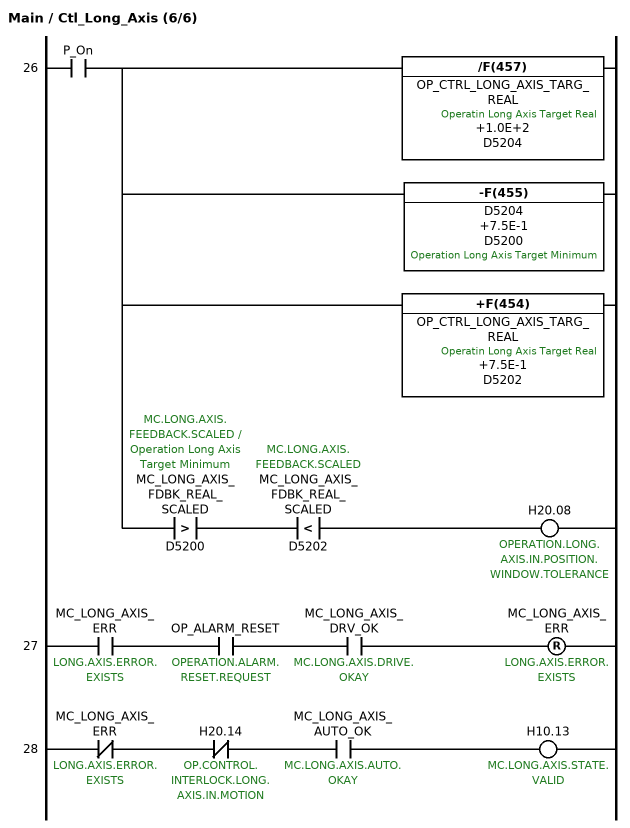
; [picture p48: Main / Ctl_Long_Axis, rungs 26-28]
; rung 26
LD P_On
/F(457) OP_CTRL_LONG_AXIS_TARG_REAL +1.0E+2 D5204  ; Operatin Long Axis Target Real
-F(455) D5204 +7.5E-1 D5200  ; Operation Long Axis Target Minimum
+F(454) OP_CTRL_LONG_AXIS_TARG_REAL +7.5E-1 D5202  ; Operatin Long Axis Target Real
AND>F(333) MC_LONG_AXIS_FDBK_REAL_SCALED D5200  ; MC.LONG.AXIS.FEEDBACK.SCALED, Operation Long Axis Target Minimum
AND<F(331) MC_LONG_AXIS_FDBK_REAL_SCALED D5202  ; MC.LONG.AXIS.FEEDBACK.SCALED
OUT H20.08  ; OPERATION.LONG.AXIS.IN.POSITION.WINDOW.TOLERANCE
; rung 27
LD MC_LONG_AXIS_ERR  ; LONG.AXIS.ERROR.EXISTS
AND OP_ALARM_RESET  ; OPERATION.ALARM.RESET.REQUEST
AND MC_LONG_AXIS_DRV_OK  ; MC.LONG.AXIS.DRIVE.OKAY
RSET MC_LONG_AXIS_ERR  ; LONG.AXIS.ERROR.EXISTS
; rung 28
LDNOT MC_LONG_AXIS_ERR  ; LONG.AXIS.ERROR.EXISTS
ANDNOT H20.14  ; OP.CONTROL.INTERLOCK.LONG.AXIS.IN.MOTION
AND MC_LONG_AXIS_AUTO_OK  ; MC.LONG.AXIS.AUTO.OKAY
OUT H10.13  ; MC.LONG.AXIS.STATE.VALID

### Section Ctl_Vertical_Axis

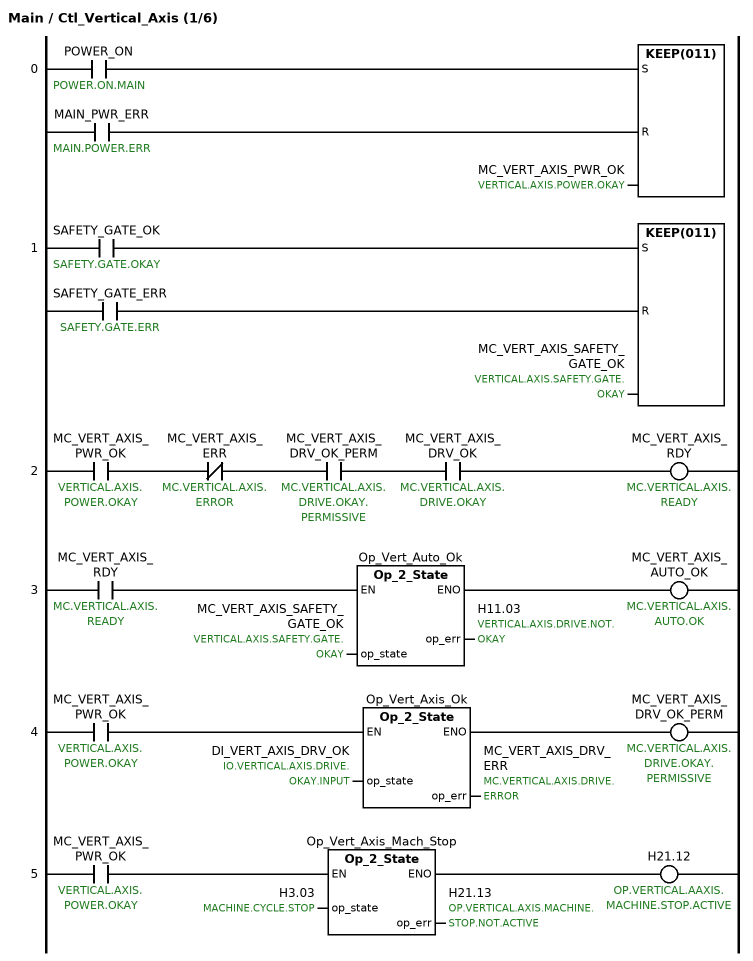
; rung 0
LD POWER_ON  ; POWER.ON.MAIN
LD MAIN_PWR_ERR  ; MAIN.POWER.ERR
KEEP(011) MC_VERT_AXIS_PWR_OK  ; VERTICAL.AXIS.POWER.OKAY
; rung 1
LD SAFETY_GATE_OK  ; SAFETY.GATE.OKAY
LD SAFETY_GATE_ERR  ; SAFETY.GATE.ERR
KEEP(011) MC_VERT_AXIS_SAFETY_GATE_OK  ; VERTICAL.AXIS.SAFETY.GATE.OKAY
; rung 2
LD MC_VERT_AXIS_PWR_OK  ; VERTICAL.AXIS.POWER.OKAY
ANDNOT MC_VERT_AXIS_ERR  ; MC.VERTICAL.AXIS.ERROR
AND MC_VERT_AXIS_DRV_OK_PERM  ; MC.VERTICAL.AXIS.DRIVE.OKAY.PERMISSIVE
AND MC_VERT_AXIS_DRV_OK  ; MC.VERTICAL.AXIS.DRIVE.OKAY
OUT MC_VERT_AXIS_RDY  ; MC.VERTICAL.AXIS.READY
; rung 3
LD MC_VERT_AXIS_RDY  ; MC.VERTICAL.AXIS.READY
CALL Op_Vert_Auto_Ok : Op_2_State (op_state := MC_VERT_AXIS_SAFETY_GATE_OK, op_err => H11.03)  ; VERTICAL.AXIS.SAFETY.GATE.OKAY, VERTICAL.AXIS.DRIVE.NOT.OKAY
OUT MC_VERT_AXIS_AUTO_OK  ; MC.VERTICAL.AXIS.AUTO.OK
; rung 4
LD MC_VERT_AXIS_PWR_OK  ; VERTICAL.AXIS.POWER.OKAY
CALL Op_Vert_Axis_Ok : Op_2_State (op_state := DI_VERT_AXIS_DRV_OK, op_err => MC_VERT_AXIS_DRV_ERR)  ; IO.VERTICAL.AXIS.DRIVE.OKAY.INPUT, MC.VERTICAL.AXIS.DRIVE.ERROR
OUT MC_VERT_AXIS_DRV_OK_PERM  ; MC.VERTICAL.AXIS.DRIVE.OKAY.PERMISSIVE
; rung 5
LD MC_VERT_AXIS_PWR_OK  ; VERTICAL.AXIS.POWER.OKAY
CALL Op_Vert_Axis_Mach_Stop : Op_2_State (op_state := H3.03, op_err => H21.13)  ; MACHINE.CYCLE.STOP, OP.VERTICAL.AXIS.MACHINE.STOP.NOT.ACTIVE
OUT H21.12  ; OP.VERTICAL.AAXIS.MACHINE.STOP.ACTIVE

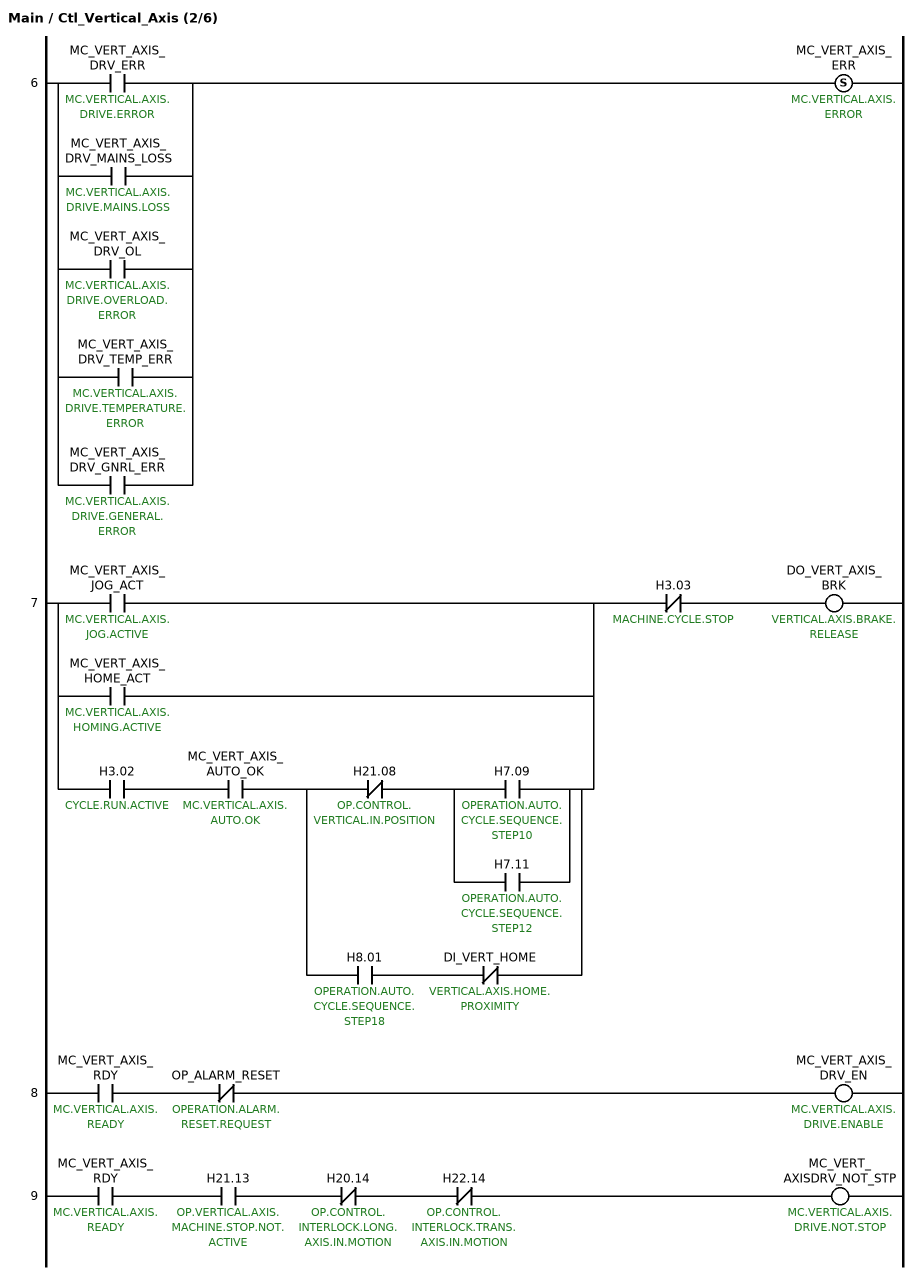
; rung 6
LD MC_VERT_AXIS_DRV_ERR  ; MC.VERTICAL.AXIS.DRIVE.ERROR
OR MC_VERT_AXIS_DRV_MAINS_LOSS  ; MC.VERTICAL.AXIS.DRIVE.MAINS.LOSS
OR MC_VERT_AXIS_DRV_OL  ; MC.VERTICAL.AXIS.DRIVE.OVERLOAD.ERROR
OR MC_VERT_AXIS_DRV_TEMP_ERR  ; MC.VERTICAL.AXIS.DRIVE.TEMPERATURE.ERROR
OR MC_VERT_AXIS_DRV_GNRL_ERR  ; MC.VERTICAL.AXIS.DRIVE.GENERAL.ERROR
SET MC_VERT_AXIS_ERR  ; MC.VERTICAL.AXIS.ERROR
; rung 7
LD MC_VERT_AXIS_JOG_ACT  ; MC.VERTICAL.AXIS.JOG.ACTIVE
OR MC_VERT_AXIS_HOME_ACT  ; MC.VERTICAL.AXIS.HOMING.ACTIVE
LD H3.02  ; CYCLE.RUN.ACTIVE
AND MC_VERT_AXIS_AUTO_OK  ; MC.VERTICAL.AXIS.AUTO.OK
LDNOT H21.08  ; OP.CONTROL.VERTICAL.IN.POSITION
LD H7.09  ; OPERATION.AUTO.CYCLE.SEQUENCE.STEP10
OR H7.11  ; OPERATION.AUTO.CYCLE.SEQUENCE.STEP12
ANDLD
LD H8.01  ; OPERATION.AUTO.CYCLE.SEQUENCE.STEP18
ANDNOT DI_VERT_HOME  ; VERTICAL.AXIS.HOME.PROXIMITY
ORLD
ANDLD
ORLD
ANDNOT H3.03  ; MACHINE.CYCLE.STOP
OUT DO_VERT_AXIS_BRK  ; VERTICAL.AXIS.BRAKE.RELEASE
; rung 8
LD MC_VERT_AXIS_RDY  ; MC.VERTICAL.AXIS.READY
ANDNOT OP_ALARM_RESET  ; OPERATION.ALARM.RESET.REQUEST
OUT MC_VERT_AXIS_DRV_EN  ; MC.VERTICAL.AXIS.DRIVE.ENABLE
; rung 9
LD MC_VERT_AXIS_RDY  ; MC.VERTICAL.AXIS.READY
AND H21.13  ; OP.VERTICAL.AXIS.MACHINE.STOP.NOT.ACTIVE
ANDNOT H20.14  ; OP.CONTROL.INTERLOCK.LONG.AXIS.IN.MOTION
ANDNOT H22.14  ; OP.CONTROL.INTERLOCK.TRANS.AXIS.IN.MOTION
OUT MC_VERT_AXISDRV_NOT_STP  ; MC.VERTICAL.AXIS.DRIVE.NOT.STOP

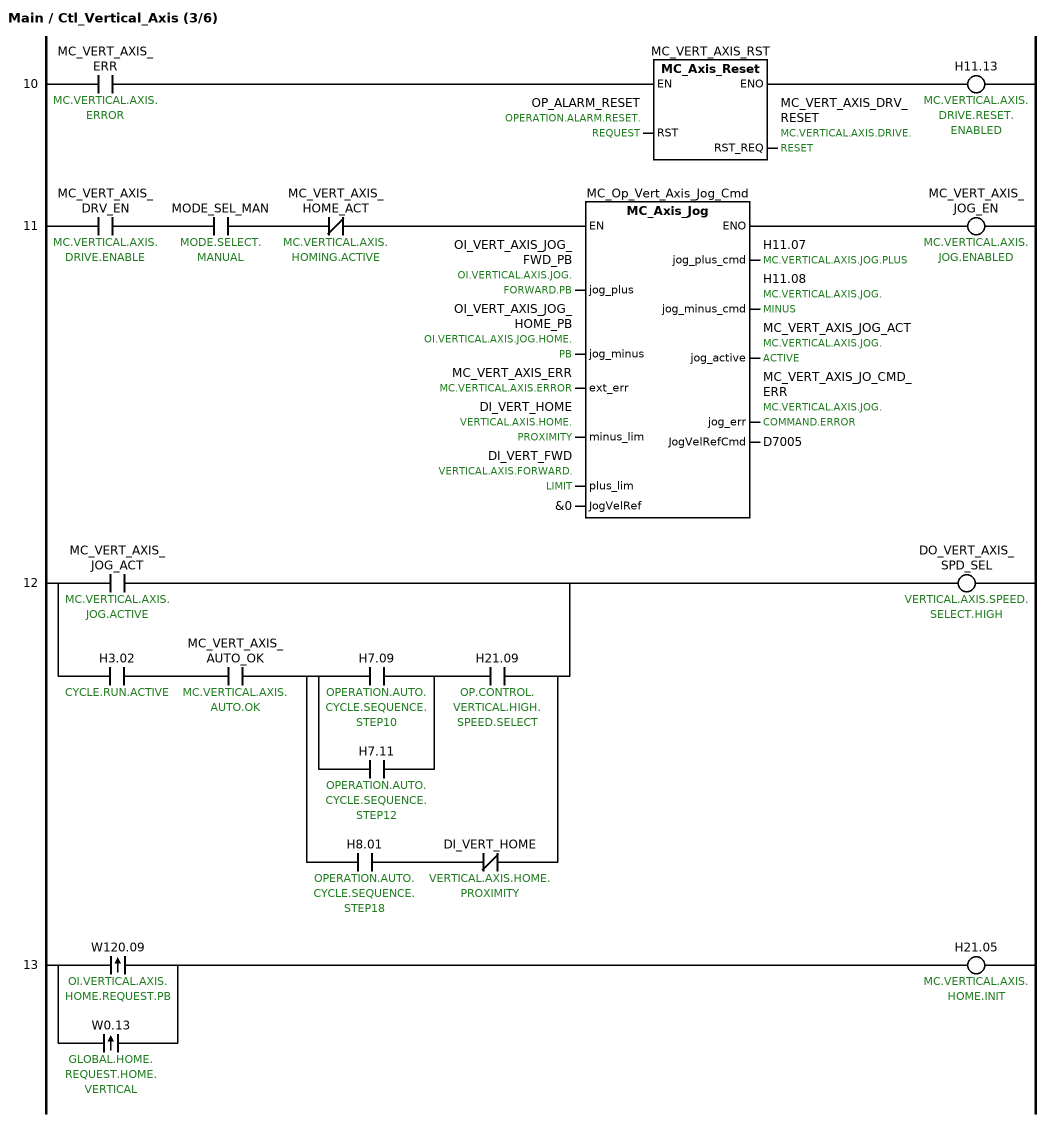
; rung 10
LD MC_VERT_AXIS_ERR  ; MC.VERTICAL.AXIS.ERROR
CALL MC_VERT_AXIS_RST : MC_Axis_Reset (RST := OP_ALARM_RESET, RST_REQ => MC_VERT_AXIS_DRV_RESET)  ; OPERATION.ALARM.RESET.REQUEST, MC.VERTICAL.AXIS.DRIVE.RESET
OUT H11.13  ; MC.VERTICAL.AXIS.DRIVE.RESET.ENABLED
; rung 11
LD MC_VERT_AXIS_DRV_EN  ; MC.VERTICAL.AXIS.DRIVE.ENABLE
AND MODE_SEL_MAN  ; MODE.SELECT.MANUAL
ANDNOT MC_VERT_AXIS_HOME_ACT  ; MC.VERTICAL.AXIS.HOMING.ACTIVE
CALL MC_Op_Vert_Axis_Jog_Cmd : MC_Axis_Jog (jog_plus := OI_VERT_AXIS_JOG_FWD_PB, jog_minus := OI_VERT_AXIS_JOG_HOME_PB, ext_err := MC_VERT_AXIS_ERR, minus_lim := DI_VERT_HOME, plus_lim := DI_VERT_FWD, JogVelRef := &0, jog_plus_cmd => H11.07, jog_minus_cmd => H11.08, jog_active => MC_VERT_AXIS_JOG_ACT, jog_err => MC_VERT_AXIS_JO_CMD_ERR, JogVelRefCmd => D7005)  ; OI.VERTICAL.AXIS.JOG.FORWARD.PB, OI.VERTICAL.AXIS.JOG.HOME.PB, MC.VERTICAL.AXIS.ERROR, VERTICAL.AXIS.HOME.PROXIMITY, VERTICAL.AXIS.FORWARD.LIMIT, MC.VERTICAL.AXIS.JOG.PLUS, MC.VERTICAL.AXIS.JOG.MINUS, MC.VERTICAL.AXIS.JOG.ACTIVE, MC.VERTICAL.AXIS.JOG.COMMAND.ERROR
OUT MC_VERT_AXIS_JOG_EN  ; MC.VERTICAL.AXIS.JOG.ENABLED
; rung 12
LD MC_VERT_AXIS_JOG_ACT  ; MC.VERTICAL.AXIS.JOG.ACTIVE
LD H3.02  ; CYCLE.RUN.ACTIVE
AND MC_VERT_AXIS_AUTO_OK  ; MC.VERTICAL.AXIS.AUTO.OK
LD H7.09  ; OPERATION.AUTO.CYCLE.SEQUENCE.STEP10
OR H7.11  ; OPERATION.AUTO.CYCLE.SEQUENCE.STEP12
AND H21.09  ; OP.CONTROL.VERTICAL.HIGH.SPEED.SELECT
LD H8.01  ; OPERATION.AUTO.CYCLE.SEQUENCE.STEP18
ANDNOT DI_VERT_HOME  ; VERTICAL.AXIS.HOME.PROXIMITY
ORLD
ANDLD
ORLD
OUT DO_VERT_AXIS_SPD_SEL  ; VERTICAL.AXIS.SPEED.SELECT.HIGH
; rung 13
@LD W120.09  ; OI.VERTICAL.AXIS.HOME.REQUEST.PB
@OR W0.13  ; GLOBAL.HOME.REQUEST.HOME.VERTICAL
OUT H21.05  ; MC.VERTICAL.AXIS.HOME.INIT

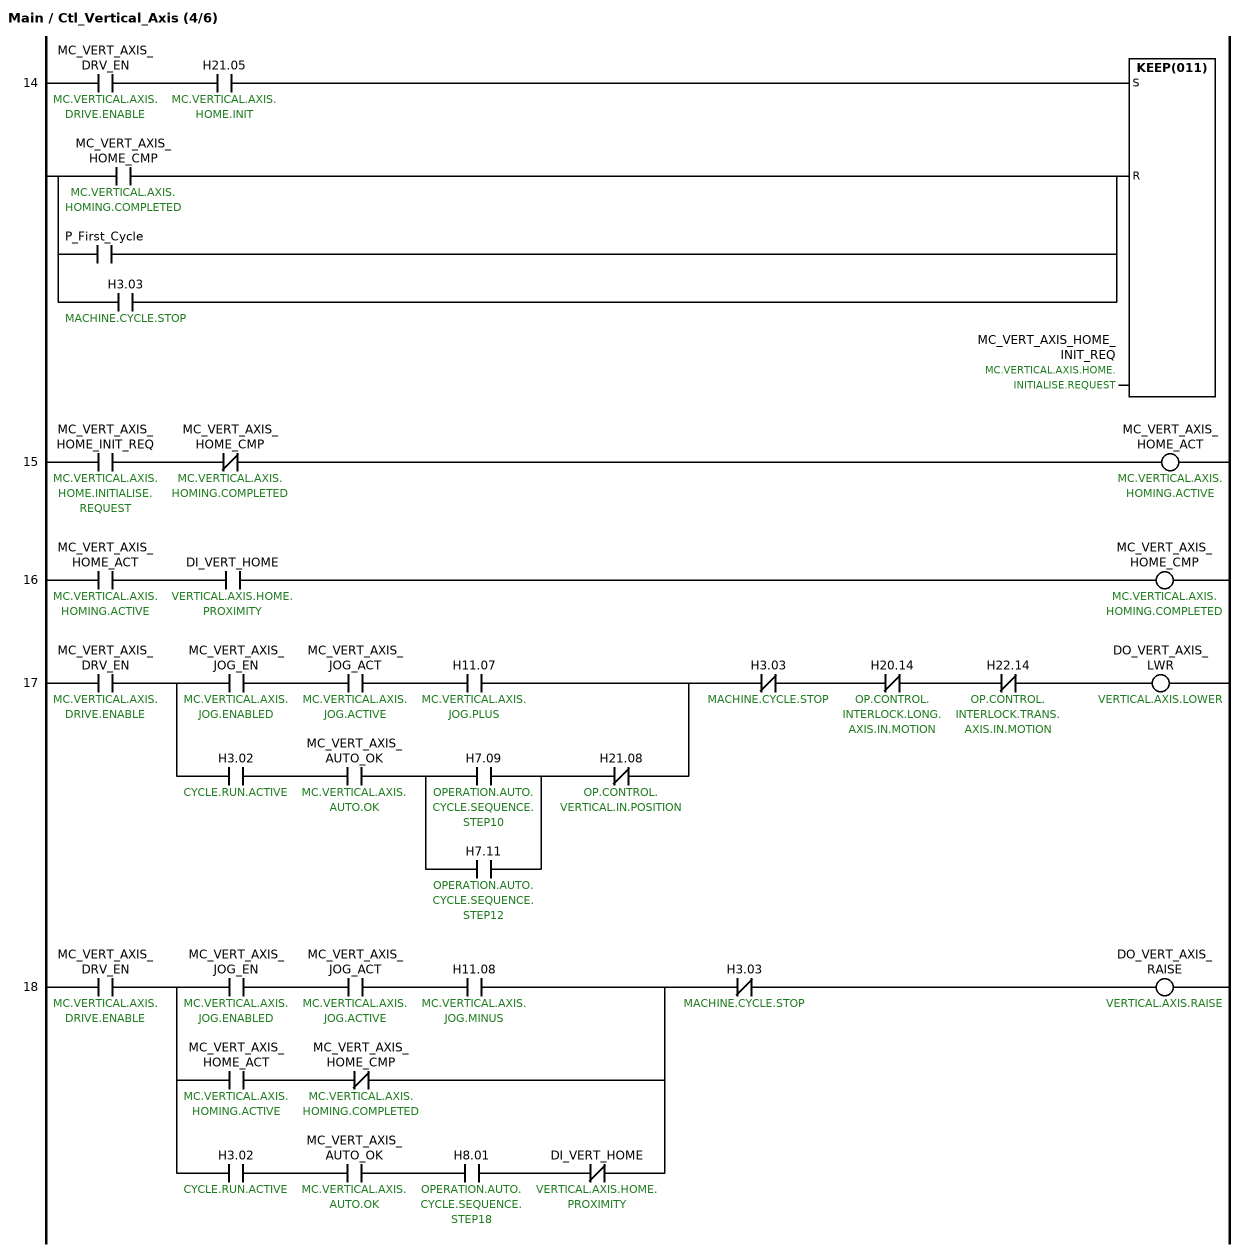
; rung 14
LD MC_VERT_AXIS_DRV_EN  ; MC.VERTICAL.AXIS.DRIVE.ENABLE
AND H21.05  ; MC.VERTICAL.AXIS.HOME.INIT
LD MC_VERT_AXIS_HOME_CMP  ; MC.VERTICAL.AXIS.HOMING.COMPLETED
OR P_First_Cycle
OR H3.03  ; MACHINE.CYCLE.STOP
KEEP(011) MC_VERT_AXIS_HOME_INIT_REQ  ; MC.VERTICAL.AXIS.HOME.INITIALISE.REQUEST
; rung 15
LD MC_VERT_AXIS_HOME_INIT_REQ  ; MC.VERTICAL.AXIS.HOME.INITIALISE.REQUEST
ANDNOT MC_VERT_AXIS_HOME_CMP  ; MC.VERTICAL.AXIS.HOMING.COMPLETED
OUT MC_VERT_AXIS_HOME_ACT  ; MC.VERTICAL.AXIS.HOMING.ACTIVE
; rung 16
LD MC_VERT_AXIS_HOME_ACT  ; MC.VERTICAL.AXIS.HOMING.ACTIVE
AND DI_VERT_HOME  ; VERTICAL.AXIS.HOME.PROXIMITY
OUT MC_VERT_AXIS_HOME_CMP  ; MC.VERTICAL.AXIS.HOMING.COMPLETED
; rung 17
LD MC_VERT_AXIS_DRV_EN  ; MC.VERTICAL.AXIS.DRIVE.ENABLE
LD MC_VERT_AXIS_JOG_EN  ; MC.VERTICAL.AXIS.JOG.ENABLED
AND MC_VERT_AXIS_JOG_ACT  ; MC.VERTICAL.AXIS.JOG.ACTIVE
AND H11.07  ; MC.VERTICAL.AXIS.JOG.PLUS
LD H3.02  ; CYCLE.RUN.ACTIVE
AND MC_VERT_AXIS_AUTO_OK  ; MC.VERTICAL.AXIS.AUTO.OK
LD H7.09  ; OPERATION.AUTO.CYCLE.SEQUENCE.STEP10
OR H7.11  ; OPERATION.AUTO.CYCLE.SEQUENCE.STEP12
ANDLD
ANDNOT H21.08  ; OP.CONTROL.VERTICAL.IN.POSITION
ORLD
ANDLD
ANDNOT H3.03  ; MACHINE.CYCLE.STOP
ANDNOT H20.14  ; OP.CONTROL.INTERLOCK.LONG.AXIS.IN.MOTION
ANDNOT H22.14  ; OP.CONTROL.INTERLOCK.TRANS.AXIS.IN.MOTION
OUT DO_VERT_AXIS_LWR  ; VERTICAL.AXIS.LOWER
; rung 18
LD MC_VERT_AXIS_DRV_EN  ; MC.VERTICAL.AXIS.DRIVE.ENABLE
LD MC_VERT_AXIS_JOG_EN  ; MC.VERTICAL.AXIS.JOG.ENABLED
AND MC_VERT_AXIS_JOG_ACT  ; MC.VERTICAL.AXIS.JOG.ACTIVE
AND H11.08  ; MC.VERTICAL.AXIS.JOG.MINUS
LD MC_VERT_AXIS_HOME_ACT  ; MC.VERTICAL.AXIS.HOMING.ACTIVE
ANDNOT MC_VERT_AXIS_HOME_CMP  ; MC.VERTICAL.AXIS.HOMING.COMPLETED
ORLD
LD H3.02  ; CYCLE.RUN.ACTIVE
AND MC_VERT_AXIS_AUTO_OK  ; MC.VERTICAL.AXIS.AUTO.OK
AND H8.01  ; OPERATION.AUTO.CYCLE.SEQUENCE.STEP18
ANDNOT DI_VERT_HOME  ; VERTICAL.AXIS.HOME.PROXIMITY
ORLD
ANDLD
ANDNOT H3.03  ; MACHINE.CYCLE.STOP
OUT DO_VERT_AXIS_RAISE  ; VERTICAL.AXIS.RAISE

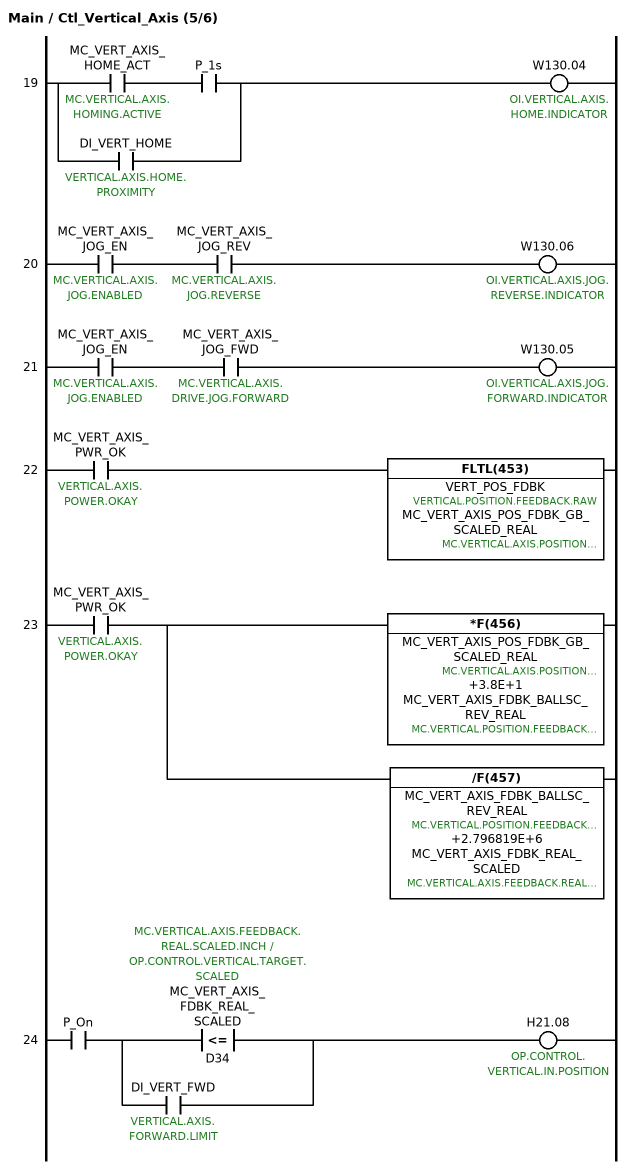
; rung 19
LD MC_VERT_AXIS_HOME_ACT  ; MC.VERTICAL.AXIS.HOMING.ACTIVE
AND P_1s
OR DI_VERT_HOME  ; VERTICAL.AXIS.HOME.PROXIMITY
OUT W130.04  ; OI.VERTICAL.AXIS.HOME.INDICATOR
; rung 20
LD MC_VERT_AXIS_JOG_EN  ; MC.VERTICAL.AXIS.JOG.ENABLED
AND MC_VERT_AXIS_JOG_REV  ; MC.VERTICAL.AXIS.JOG.REVERSE
OUT W130.06  ; OI.VERTICAL.AXIS.JOG.REVERSE.INDICATOR
; rung 21
LD MC_VERT_AXIS_JOG_EN  ; MC.VERTICAL.AXIS.JOG.ENABLED
AND MC_VERT_AXIS_JOG_FWD  ; MC.VERTICAL.AXIS.DRIVE.JOG.FORWARD
OUT W130.05  ; OI.VERTICAL.AXIS.JOG.FORWARD.INDICATOR
; rung 22
LD MC_VERT_AXIS_PWR_OK  ; VERTICAL.AXIS.POWER.OKAY
FLTL(453) VERT_POS_FDBK MC_VERT_AXIS_POS_FDBK_GB_SCALED_REAL  ; VERTICAL.POSITION.FEEDBACK.RAW, MC.VERTICAL.AXIS.POSITION.REVOLUTION.REAL
; rung 23
LD MC_VERT_AXIS_PWR_OK  ; VERTICAL.AXIS.POWER.OKAY
*F(456) MC_VERT_AXIS_POS_FDBK_GB_SCALED_REAL +3.8E+1 MC_VERT_AXIS_FDBK_BALLSC_REV_REAL  ; MC.VERTICAL.AXIS.POSITION.REVOLUTION.REAL, MC.VERTICAL.POSITION.FEEDBACK.BALLSCREW.REVOLUTIONS.REAL
/F(457) MC_VERT_AXIS_FDBK_BALLSC_REV_REAL +2.796819E+6 MC_VERT_AXIS_FDBK_REAL_SCALED  ; MC.VERTICAL.POSITION.FEEDBACK.BALLSCREW.REVOLUTIONS.REAL, MC.VERTICAL.AXIS.FEEDBACK.REAL.SCALED.INCH
; rung 24
LD P_On
LD<=F(332) MC_VERT_AXIS_FDBK_REAL_SCALED D34  ; MC.VERTICAL.AXIS.FEEDBACK.REAL.SCALED.INCH, OP.CONTROL.VERTICAL.TARGET.SCALED
OR DI_VERT_FWD  ; VERTICAL.AXIS.FORWARD.LIMIT
ANDLD
OUT H21.08  ; OP.CONTROL.VERTICAL.IN.POSITION

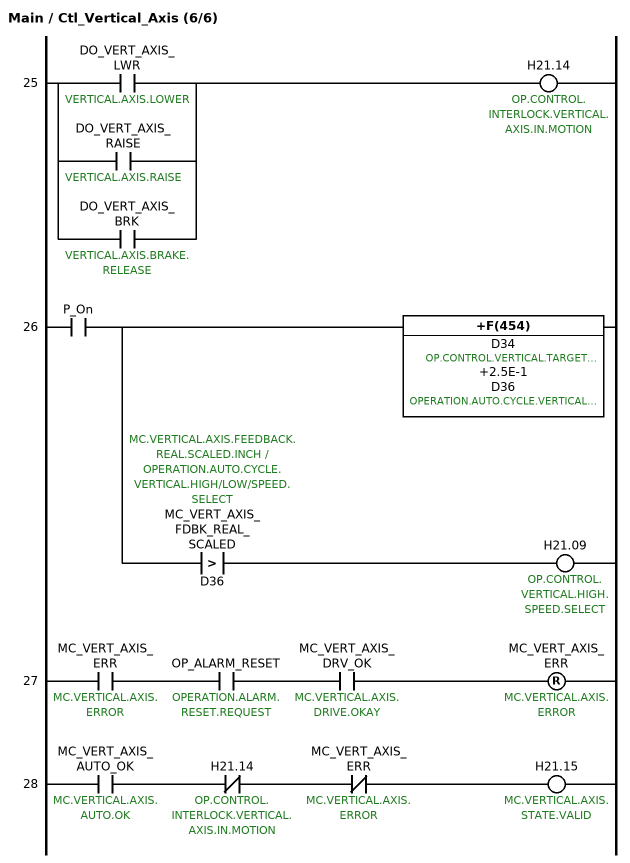
; rung 25
LD DO_VERT_AXIS_LWR  ; VERTICAL.AXIS.LOWER
OR DO_VERT_AXIS_RAISE  ; VERTICAL.AXIS.RAISE
OR DO_VERT_AXIS_BRK  ; VERTICAL.AXIS.BRAKE.RELEASE
OUT H21.14  ; OP.CONTROL.INTERLOCK.VERTICAL.AXIS.IN.MOTION
; rung 26
LD P_On
+F(454) D34 +2.5E-1 D36  ; OP.CONTROL.VERTICAL.TARGET.SCALED, OPERATION.AUTO.CYCLE.VERTICAL.HIGH/LOW/SPEED.SELECT
AND>F(333) MC_VERT_AXIS_FDBK_REAL_SCALED D36  ; MC.VERTICAL.AXIS.FEEDBACK.REAL.SCALED.INCH, OPERATION.AUTO.CYCLE.VERTICAL.HIGH/LOW/SPEED.SELECT
OUT H21.09  ; OP.CONTROL.VERTICAL.HIGH.SPEED.SELECT
; rung 27
LD MC_VERT_AXIS_ERR  ; MC.VERTICAL.AXIS.ERROR
AND OP_ALARM_RESET  ; OPERATION.ALARM.RESET.REQUEST
AND MC_VERT_AXIS_DRV_OK  ; MC.VERTICAL.AXIS.DRIVE.OKAY
RSET MC_VERT_AXIS_ERR  ; MC.VERTICAL.AXIS.ERROR
; rung 28
LD MC_VERT_AXIS_AUTO_OK  ; MC.VERTICAL.AXIS.AUTO.OK
ANDNOT H21.14  ; OP.CONTROL.INTERLOCK.VERTICAL.AXIS.IN.MOTION
ANDNOT MC_VERT_AXIS_ERR  ; MC.VERTICAL.AXIS.ERROR
OUT H21.15  ; MC.VERTICAL.AXIS.STATE.VALID

### Section Ctl_Transverse_Axis

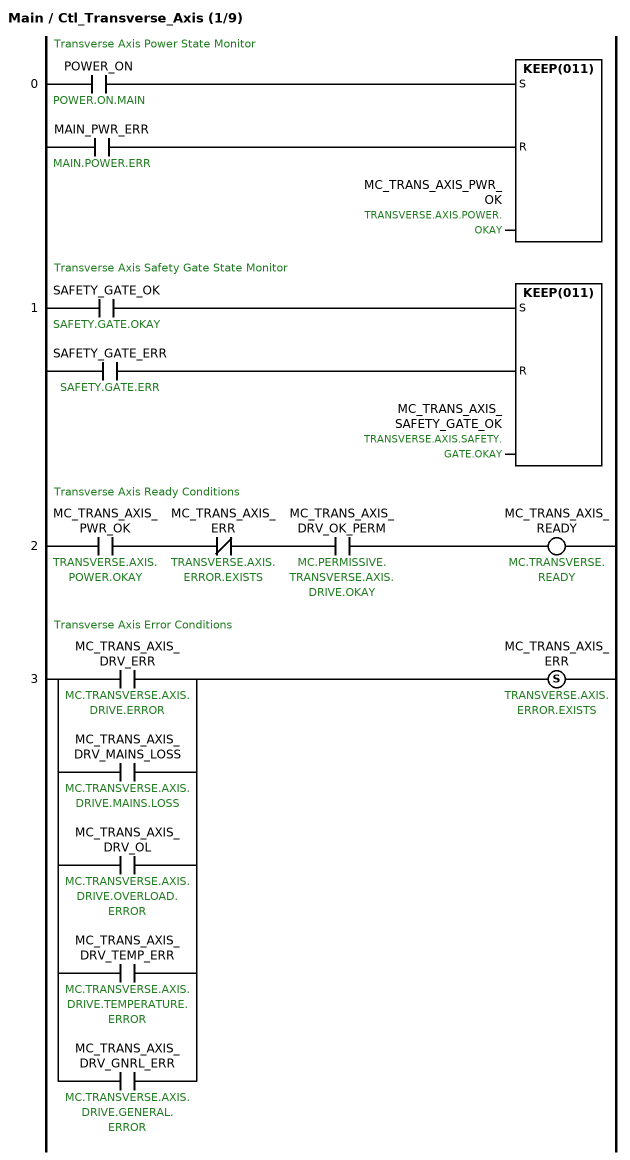
; rung 0: Transverse Axis Power State Monitor
LD POWER_ON  ; POWER.ON.MAIN
LD MAIN_PWR_ERR  ; MAIN.POWER.ERR
KEEP(011) MC_TRANS_AXIS_PWR_OK  ; TRANSVERSE.AXIS.POWER.OKAY
; rung 1: Transverse Axis Safety Gate State Monitor
LD SAFETY_GATE_OK  ; SAFETY.GATE.OKAY
LD SAFETY_GATE_ERR  ; SAFETY.GATE.ERR
KEEP(011) MC_TRANS_AXIS_SAFETY_GATE_OK  ; TRANSVERSE.AXIS.SAFETY.GATE.OKAY
; rung 2: Transverse Axis Ready Conditions
LD MC_TRANS_AXIS_PWR_OK  ; TRANSVERSE.AXIS.POWER.OKAY
ANDNOT MC_TRANS_AXIS_ERR  ; TRANSVERSE.AXIS.ERROR.EXISTS
AND MC_TRANS_AXIS_DRV_OK_PERM  ; MC.PERMISSIVE.TRANSVERSE.AXIS.DRIVE.OKAY
OUT MC_TRANS_AXIS_READY  ; MC.TRANSVERSE.READY
; rung 3: Transverse Axis Error Conditions
LD MC_TRANS_AXIS_DRV_ERR  ; MC.TRANSVERSE.AXIS.DRIVE.ERROR
OR MC_TRANS_AXIS_DRV_MAINS_LOSS  ; MC.TRANSVERSE.AXIS.DRIVE.MAINS.LOSS
OR MC_TRANS_AXIS_DRV_OL  ; MC.TRANSVERSE.AXIS.DRIVE.OVERLOAD.ERROR
OR MC_TRANS_AXIS_DRV_TEMP_ERR  ; MC.TRANSVERSE.AXIS.DRIVE.TEMPERATURE.ERROR
OR MC_TRANS_AXIS_DRV_GNRL_ERR  ; MC.TRANSVERSE.AXIS.DRIVE.GENERAL.ERROR
SET MC_TRANS_AXIS_ERR  ; TRANSVERSE.AXIS.ERROR.EXISTS

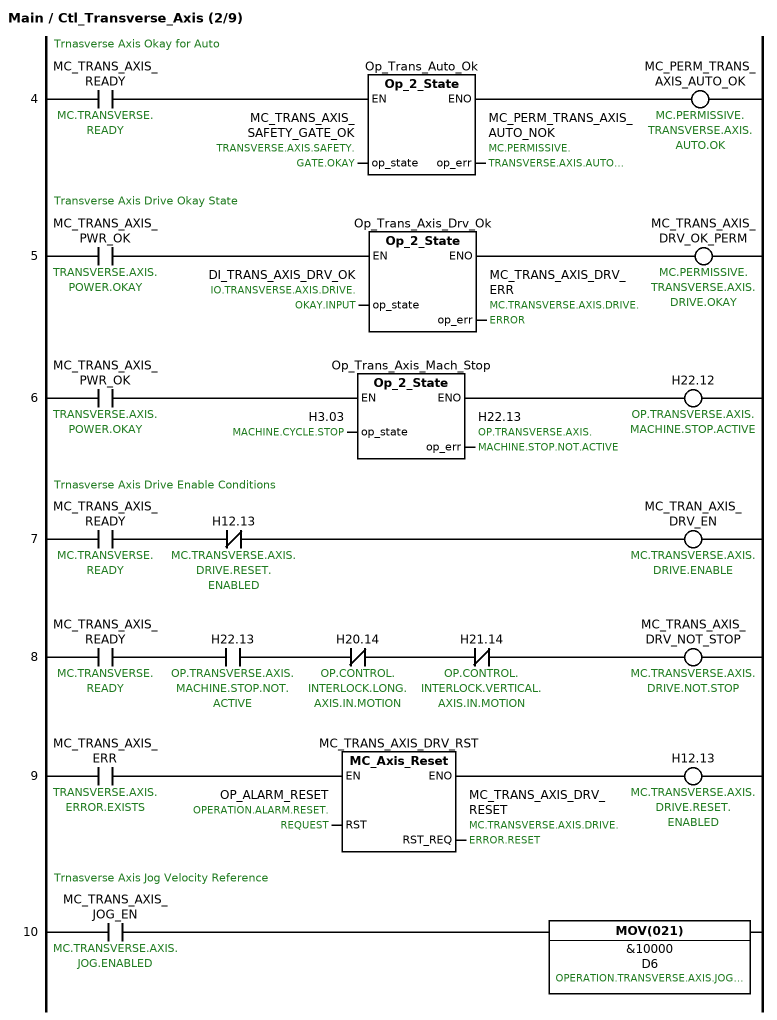
; rung 4: Trnasverse Axis Okay for Auto
LD MC_TRANS_AXIS_READY  ; MC.TRANSVERSE.READY
CALL Op_Trans_Auto_Ok : Op_2_State (op_state := MC_TRANS_AXIS_SAFETY_GATE_OK, op_err => MC_PERM_TRANS_AXIS_AUTO_NOK)  ; TRANSVERSE.AXIS.SAFETY.GATE.OKAY, MC.PERMISSIVE.TRANSVERSE.AXIS.AUTO.NOK
OUT MC_PERM_TRANS_AXIS_AUTO_OK  ; MC.PERMISSIVE.TRANSVERSE.AXIS.AUTO.OK
; rung 5: Transverse Axis Drive Okay State
LD MC_TRANS_AXIS_PWR_OK  ; TRANSVERSE.AXIS.POWER.OKAY
CALL Op_Trans_Axis_Drv_Ok : Op_2_State (op_state := DI_TRANS_AXIS_DRV_OK, op_err => MC_TRANS_AXIS_DRV_ERR)  ; IO.TRANSVERSE.AXIS.DRIVE.OKAY.INPUT, MC.TRANSVERSE.AXIS.DRIVE.ERROR
OUT MC_TRANS_AXIS_DRV_OK_PERM  ; MC.PERMISSIVE.TRANSVERSE.AXIS.DRIVE.OKAY
; rung 6
LD MC_TRANS_AXIS_PWR_OK  ; TRANSVERSE.AXIS.POWER.OKAY
CALL Op_Trans_Axis_Mach_Stop : Op_2_State (op_state := H3.03, op_err => H22.13)  ; MACHINE.CYCLE.STOP, OP.TRANSVERSE.AXIS.MACHINE.STOP.NOT.ACTIVE
OUT H22.12  ; OP.TRANSVERSE.AXIS.MACHINE.STOP.ACTIVE
; rung 7: Trnasverse Axis Drive Enable Conditions
LD MC_TRANS_AXIS_READY  ; MC.TRANSVERSE.READY
ANDNOT H12.13  ; MC.TRANSVERSE.AXIS.DRIVE.RESET.ENABLED
OUT MC_TRAN_AXIS_DRV_EN  ; MC.TRANSVERSE.AXIS.DRIVE.ENABLE
; rung 8
LD MC_TRANS_AXIS_READY  ; MC.TRANSVERSE.READY
AND H22.13  ; OP.TRANSVERSE.AXIS.MACHINE.STOP.NOT.ACTIVE
ANDNOT H20.14  ; OP.CONTROL.INTERLOCK.LONG.AXIS.IN.MOTION
ANDNOT H21.14  ; OP.CONTROL.INTERLOCK.VERTICAL.AXIS.IN.MOTION
OUT MC_TRANS_AXIS_DRV_NOT_STOP  ; MC.TRANSVERSE.AXIS.DRIVE.NOT.STOP
; rung 9
LD MC_TRANS_AXIS_ERR  ; TRANSVERSE.AXIS.ERROR.EXISTS
CALL MC_TRANS_AXIS_DRV_RST : MC_Axis_Reset (RST := OP_ALARM_RESET, RST_REQ => MC_TRANS_AXIS_DRV_RESET)  ; OPERATION.ALARM.RESET.REQUEST, MC.TRANSVERSE.AXIS.DRIVE.ERROR.RESET
OUT H12.13  ; MC.TRANSVERSE.AXIS.DRIVE.RESET.ENABLED
; rung 10: Trnasverse Axis Jog Velocity Reference
LD MC_TRANS_AXIS_JOG_EN  ; MC.TRANSVERSE.AXIS.JOG.ENABLED
MOV(021) &10000 D6  ; OPERATION.TRANSVERSE.AXIS.JOG.VELOCITY.REFERNCE.WORD

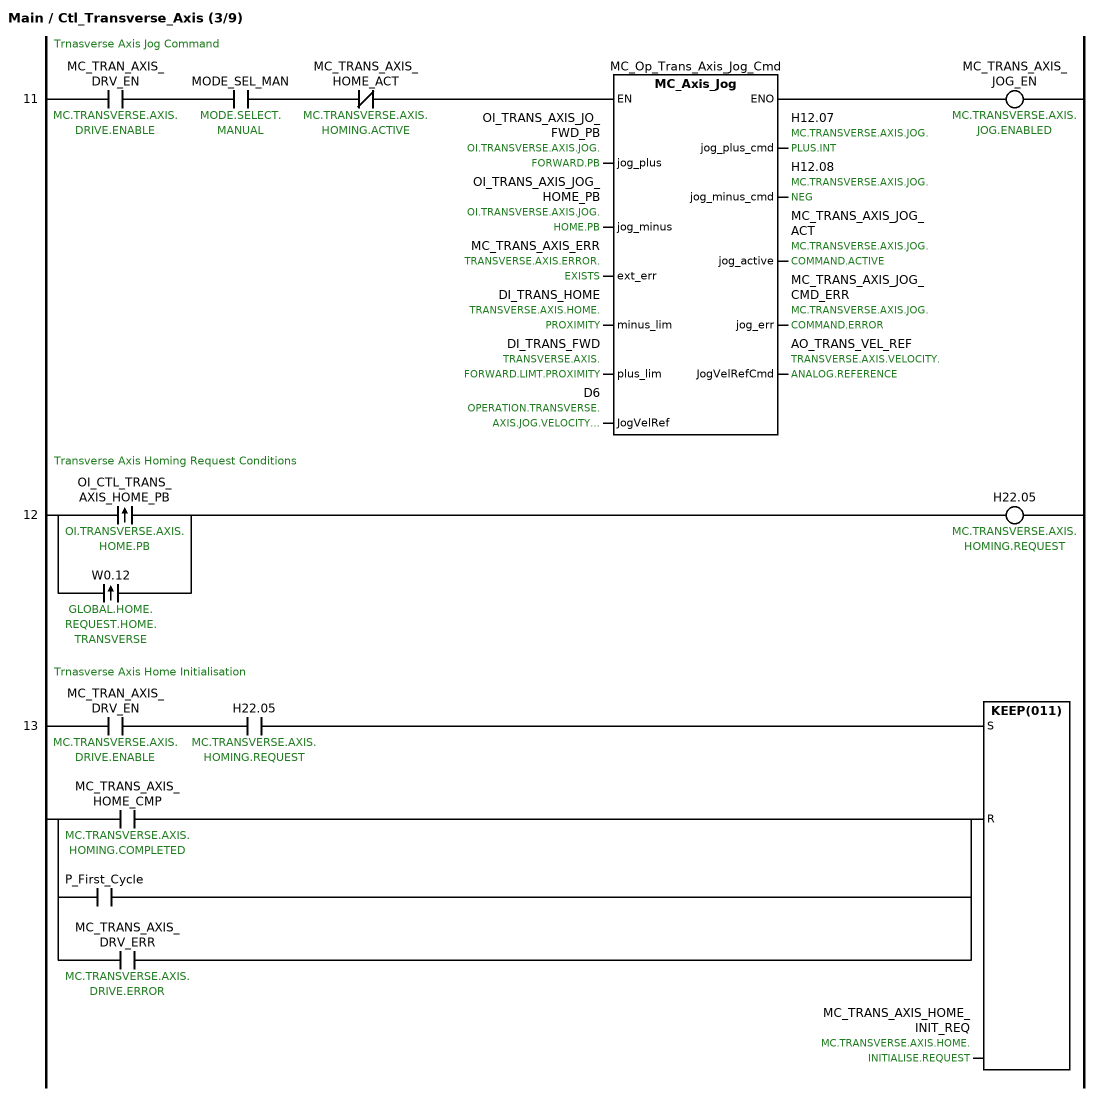
; rung 11: Trnasverse Axis Jog Command
LD MC_TRAN_AXIS_DRV_EN  ; MC.TRANSVERSE.AXIS.DRIVE.ENABLE
AND MODE_SEL_MAN  ; MODE.SELECT.MANUAL
ANDNOT MC_TRANS_AXIS_HOME_ACT  ; MC.TRANSVERSE.AXIS.HOMING.ACTIVE
CALL MC_Op_Trans_Axis_Jog_Cmd : MC_Axis_Jog (jog_plus := OI_TRANS_AXIS_JO_FWD_PB, jog_minus := OI_TRANS_AXIS_JOG_HOME_PB, ext_err := MC_TRANS_AXIS_ERR, minus_lim := DI_TRANS_HOME, plus_lim := DI_TRANS_FWD, JogVelRef := D6, jog_plus_cmd => H12.07, jog_minus_cmd => H12.08, jog_active => MC_TRANS_AXIS_JOG_ACT, jog_err => MC_TRANS_AXIS_JOG_CMD_ERR, JogVelRefCmd => AO_TRANS_VEL_REF)  ; OI.TRANSVERSE.AXIS.JOG.FORWARD.PB, OI.TRANSVERSE.AXIS.JOG.HOME.PB, TRANSVERSE.AXIS.ERROR.EXISTS, TRANSVERSE.AXIS.HOME.PROXIMITY, TRANSVERSE.AXIS.FORWARD.LIMT.PROXIMITY, OPERATION.TRANSVERSE.AXIS.JOG.VELOCITY.REFERNCE.WORD, MC.TRANSVERSE.AXIS.JOG.PLUS.INT, MC.TRANSVERSE.AXIS.JOG.NEG, MC.TRANSVERSE.AXIS.JOG.COMMAND.ACTIVE, MC.TRANSVERSE.AXIS.JOG.COMMAND.ERROR, TRANSVERSE.AXIS.VELOCITY.ANALOG.REFERENCE
OUT MC_TRANS_AXIS_JOG_EN  ; MC.TRANSVERSE.AXIS.JOG.ENABLED
; rung 12: Transverse Axis Homing Request Conditions
@LD OI_CTL_TRANS_AXIS_HOME_PB  ; OI.TRANSVERSE.AXIS.HOME.PB
@OR W0.12  ; GLOBAL.HOME.REQUEST.HOME.TRANSVERSE
OUT H22.05  ; MC.TRANSVERSE.AXIS.HOMING.REQUEST
; rung 13: Trnasverse Axis Home Initialisation
LD MC_TRAN_AXIS_DRV_EN  ; MC.TRANSVERSE.AXIS.DRIVE.ENABLE
AND H22.05  ; MC.TRANSVERSE.AXIS.HOMING.REQUEST
LD MC_TRANS_AXIS_HOME_CMP  ; MC.TRANSVERSE.AXIS.HOMING.COMPLETED
OR P_First_Cycle
OR MC_TRANS_AXIS_DRV_ERR  ; MC.TRANSVERSE.AXIS.DRIVE.ERROR
KEEP(011) MC_TRANS_AXIS_HOME_INIT_REQ  ; MC.TRANSVERSE.AXIS.HOME.INITIALISE.REQUEST

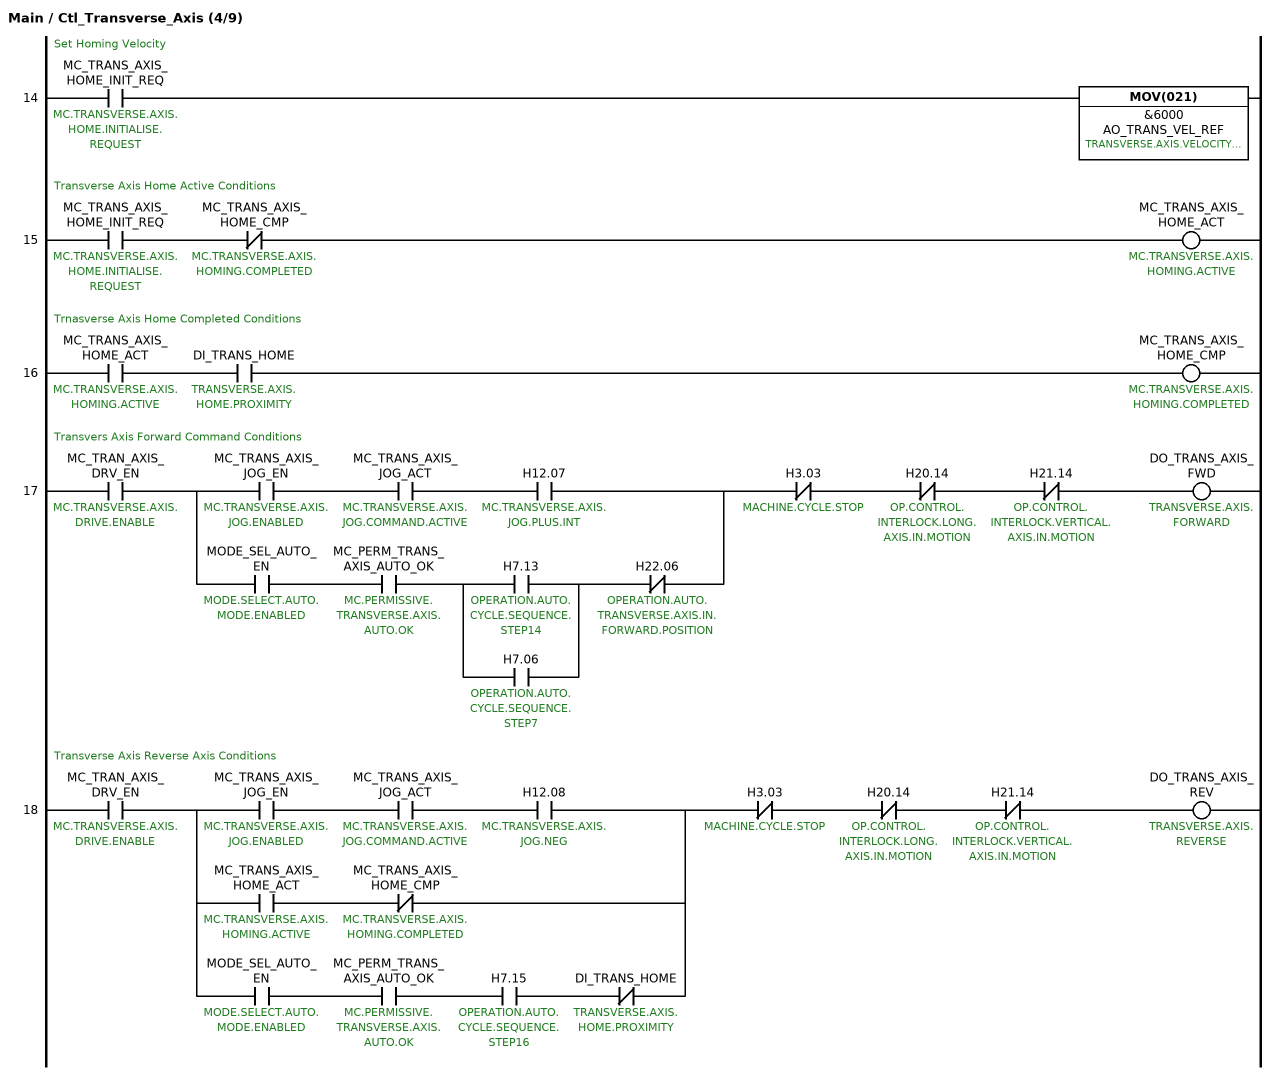
; rung 14: Set Homing Velocity
LD MC_TRANS_AXIS_HOME_INIT_REQ  ; MC.TRANSVERSE.AXIS.HOME.INITIALISE.REQUEST
MOV(021) &6000 AO_TRANS_VEL_REF  ; TRANSVERSE.AXIS.VELOCITY.ANALOG.REFERENCE
; rung 15: Transverse Axis Home Active Conditions
LD MC_TRANS_AXIS_HOME_INIT_REQ  ; MC.TRANSVERSE.AXIS.HOME.INITIALISE.REQUEST
ANDNOT MC_TRANS_AXIS_HOME_CMP  ; MC.TRANSVERSE.AXIS.HOMING.COMPLETED
OUT MC_TRANS_AXIS_HOME_ACT  ; MC.TRANSVERSE.AXIS.HOMING.ACTIVE
; rung 16: Trnasverse Axis Home Completed Conditions
LD MC_TRANS_AXIS_HOME_ACT  ; MC.TRANSVERSE.AXIS.HOMING.ACTIVE
AND DI_TRANS_HOME  ; TRANSVERSE.AXIS.HOME.PROXIMITY
OUT MC_TRANS_AXIS_HOME_CMP  ; MC.TRANSVERSE.AXIS.HOMING.COMPLETED
; rung 17: Transvers Axis Forward Command Conditions
LD MC_TRAN_AXIS_DRV_EN  ; MC.TRANSVERSE.AXIS.DRIVE.ENABLE
LD MC_TRANS_AXIS_JOG_EN  ; MC.TRANSVERSE.AXIS.JOG.ENABLED
AND MC_TRANS_AXIS_JOG_ACT  ; MC.TRANSVERSE.AXIS.JOG.COMMAND.ACTIVE
AND H12.07  ; MC.TRANSVERSE.AXIS.JOG.PLUS.INT
LD MODE_SEL_AUTO_EN  ; MODE.SELECT.AUTO.MODE.ENABLED
AND MC_PERM_TRANS_AXIS_AUTO_OK  ; MC.PERMISSIVE.TRANSVERSE.AXIS.AUTO.OK
LD H7.13  ; OPERATION.AUTO.CYCLE.SEQUENCE.STEP14
OR H7.06  ; OPERATION.AUTO.CYCLE.SEQUENCE.STEP7
ANDLD
ANDNOT H22.06  ; OPERATION.AUTO.TRANSVERSE.AXIS.IN.FORWARD.POSITION
ORLD
ANDLD
ANDNOT H3.03  ; MACHINE.CYCLE.STOP
ANDNOT H20.14  ; OP.CONTROL.INTERLOCK.LONG.AXIS.IN.MOTION
ANDNOT H21.14  ; OP.CONTROL.INTERLOCK.VERTICAL.AXIS.IN.MOTION
OUT DO_TRANS_AXIS_FWD  ; TRANSVERSE.AXIS.FORWARD
; rung 18: Transverse Axis Reverse Axis Conditions
LD MC_TRAN_AXIS_DRV_EN  ; MC.TRANSVERSE.AXIS.DRIVE.ENABLE
LD MC_TRANS_AXIS_JOG_EN  ; MC.TRANSVERSE.AXIS.JOG.ENABLED
AND MC_TRANS_AXIS_JOG_ACT  ; MC.TRANSVERSE.AXIS.JOG.COMMAND.ACTIVE
AND H12.08  ; MC.TRANSVERSE.AXIS.JOG.NEG
LD MC_TRANS_AXIS_HOME_ACT  ; MC.TRANSVERSE.AXIS.HOMING.ACTIVE
ANDNOT MC_TRANS_AXIS_HOME_CMP  ; MC.TRANSVERSE.AXIS.HOMING.COMPLETED
ORLD
LD MODE_SEL_AUTO_EN  ; MODE.SELECT.AUTO.MODE.ENABLED
AND MC_PERM_TRANS_AXIS_AUTO_OK  ; MC.PERMISSIVE.TRANSVERSE.AXIS.AUTO.OK
AND H7.15  ; OPERATION.AUTO.CYCLE.SEQUENCE.STEP16
ANDNOT DI_TRANS_HOME  ; TRANSVERSE.AXIS.HOME.PROXIMITY
ORLD
ANDLD
ANDNOT H3.03  ; MACHINE.CYCLE.STOP
ANDNOT H20.14  ; OP.CONTROL.INTERLOCK.LONG.AXIS.IN.MOTION
ANDNOT H21.14  ; OP.CONTROL.INTERLOCK.VERTICAL.AXIS.IN.MOTION
OUT DO_TRANS_AXIS_REV  ; TRANSVERSE.AXIS.REVERSE

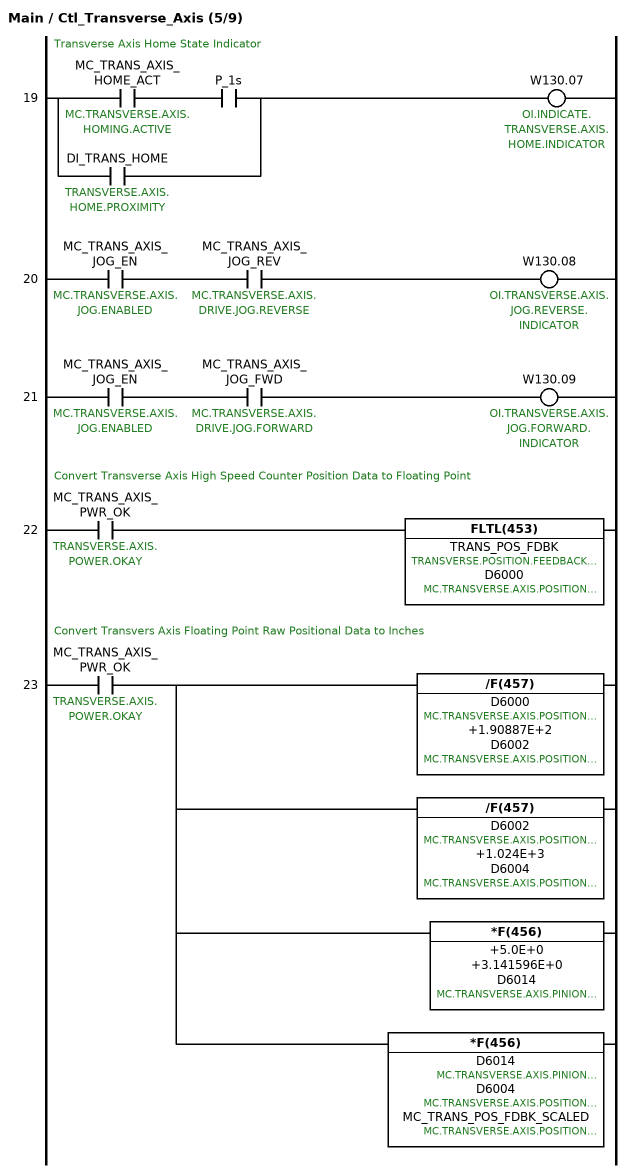
; rung 19: Transverse Axis Home State Indicator
LD MC_TRANS_AXIS_HOME_ACT  ; MC.TRANSVERSE.AXIS.HOMING.ACTIVE
AND P_1s
OR DI_TRANS_HOME  ; TRANSVERSE.AXIS.HOME.PROXIMITY
OUT W130.07  ; OI.INDICATE.TRANSVERSE.AXIS.HOME.INDICATOR
; rung 20
LD MC_TRANS_AXIS_JOG_EN  ; MC.TRANSVERSE.AXIS.JOG.ENABLED
AND MC_TRANS_AXIS_JOG_REV  ; MC.TRANSVERSE.AXIS.DRIVE.JOG.REVERSE
OUT W130.08  ; OI.TRANSVERSE.AXIS.JOG.REVERSE.INDICATOR
; rung 21
LD MC_TRANS_AXIS_JOG_EN  ; MC.TRANSVERSE.AXIS.JOG.ENABLED
AND MC_TRANS_AXIS_JOG_FWD  ; MC.TRANSVERSE.AXIS.DRIVE.JOG.FORWARD
OUT W130.09  ; OI.TRANSVERSE.AXIS.JOG.FORWARD.INDICATOR
; rung 22: Convert Transverse Axis High Speed Counter Position Data to Floating Point
LD MC_TRANS_AXIS_PWR_OK  ; TRANSVERSE.AXIS.POWER.OKAY
FLTL(453) TRANS_POS_FDBK D6000  ; TRANSVERSE.POSITION.FEEDBACK.RAW, MC.TRANSVERSE.AXIS.POSITION.FEEDBACK.RAW.REAL
; rung 23: Convert Transvers Axis Floating Point Raw Positional Data to Inches
LD MC_TRANS_AXIS_PWR_OK  ; TRANSVERSE.AXIS.POWER.OKAY
/F(457) D6000 +1.90887E+2 D6002  ; MC.TRANSVERSE.AXIS.POSITION.FEEDBACK.RAW.REAL, MC.TRANSVERSE.AXIS.POSITION.FEEDBACK.GB.SCALED.REAL
/F(457) D6002 +1.024E+3 D6004  ; MC.TRANSVERSE.AXIS.POSITION.FEEDBACK.GB.SCALED.REAL, MC.TRANSVERSE.AXIS.POSITION.PINION.REVOLUTIONS.REAL
*F(456) +5.0E+0 +3.141596E+0 D6014  ; MC.TRANSVERSE.AXIS.PINION.CIRCUMFERENCE.INCHES.REAL
*F(456) D6014 D6004 MC_TRANS_POS_FDBK_SCALED  ; MC.TRANSVERSE.AXIS.PINION.CIRCUMFERENCE.INCHES.REAL, MC.TRANSVERSE.AXIS.POSITION.PINION.REVOLUTIONS.REAL, MC.TRANSVERSE.AXIS.POSITION.FEEDBACK.INCHES.SCALED.REAL

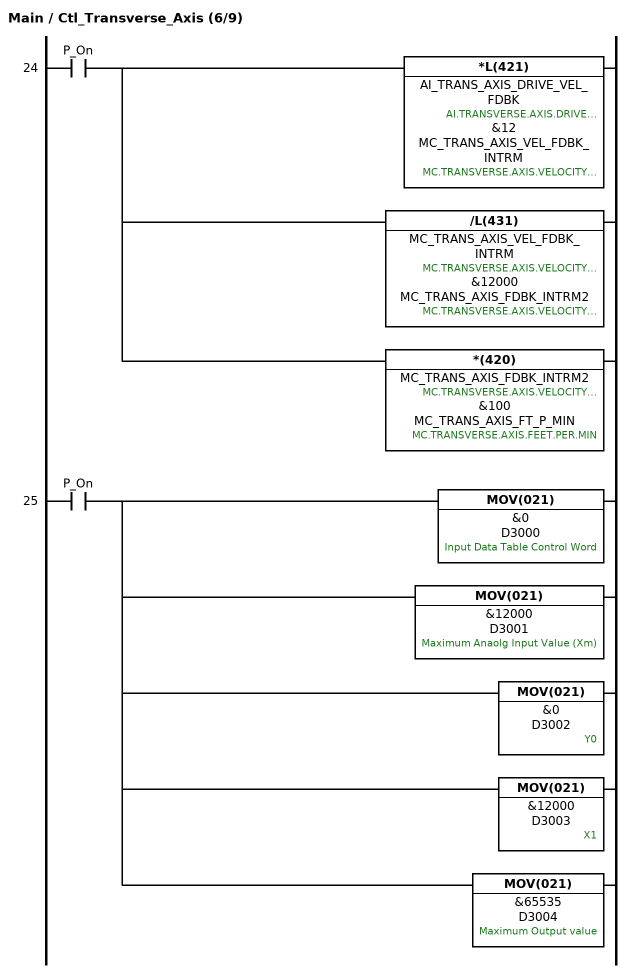
; rung 24
LD P_On
*L(421) AI_TRANS_AXIS_DRIVE_VEL_FDBK &12 MC_TRANS_AXIS_VEL_FDBK_INTRM  ; AI.TRANSVERSE.AXIS.DRIVE.VELOCITY.FEEDBACK, MC.TRANSVERSE.AXIS.VELOCITY.FEEDBACK.INTERIM
/L(431) MC_TRANS_AXIS_VEL_FDBK_INTRM &12000 MC_TRANS_AXIS_FDBK_INTRM2  ; MC.TRANSVERSE.AXIS.VELOCITY.FEEDBACK.INTERIM, MC.TRANSVERSE.AXIS.VELOCITY.FEEDBACK.INTERIM2
*(420) MC_TRANS_AXIS_FDBK_INTRM2 &100 MC_TRANS_AXIS_FT_P_MIN  ; MC.TRANSVERSE.AXIS.VELOCITY.FEEDBACK.INTERIM2, MC.TRANSVERSE.AXIS.FEET.PER.MIN
; rung 25
LD P_On
MOV(021) &0 D3000  ; Input Data Table Control Word
MOV(021) &12000 D3001  ; Maximum Anaolg Input Value (Xm)
MOV(021) &0 D3002  ; Y0
MOV(021) &12000 D3003  ; X1
MOV(021) &65535 D3004  ; Maximum Output value

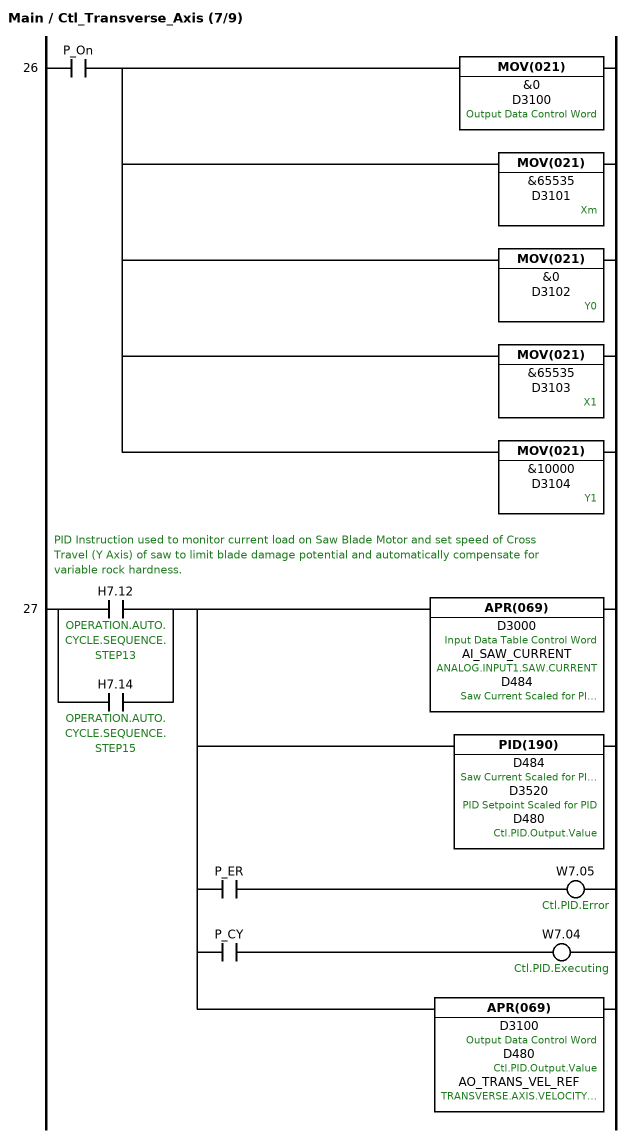
; rung 26
LD P_On
MOV(021) &0 D3100  ; Output Data Control Word
MOV(021) &65535 D3101  ; Xm
MOV(021) &0 D3102  ; Y0
MOV(021) &65535 D3103  ; X1
MOV(021) &10000 D3104  ; Y1
; rung 27: PID Instruction used to monitor current load on Saw Blade Motor and set speed of Cross Travel (Y Axis) of saw to limit blade damage potential and automatically compensate for variable rock hardness.
LD H7.12  ; OPERATION.AUTO.CYCLE.SEQUENCE.STEP13
OR H7.14  ; OPERATION.AUTO.CYCLE.SEQUENCE.STEP15
OUT TR0
APR(069) D3000 AI_SAW_CURRENT D484  ; Input Data Table Control Word, ANALOG.INPUT1.SAW.CURRENT, Saw Current Scaled for PID instruction use
PID(190) D484 D3520 D480  ; Saw Current Scaled for PID instruction use, PID Setpoint Scaled for PID, Ctl.PID.Output.Value
AND P_ER
OUT W7.05  ; Ctl.PID.Error  // Set BitW7.05 to High if PID instruction Errors
LD TR0
AND P_CY
OUT W7.04  ; Ctl.PID.Executing  // When PID is executing W7.04 is High
LD TR0
APR(069) D3100 D480 AO_TRANS_VEL_REF  ; Output Data Control Word, Ctl.PID.Output.Value, TRANSVERSE.AXIS.VELOCITY.ANALOG.REFERENCE

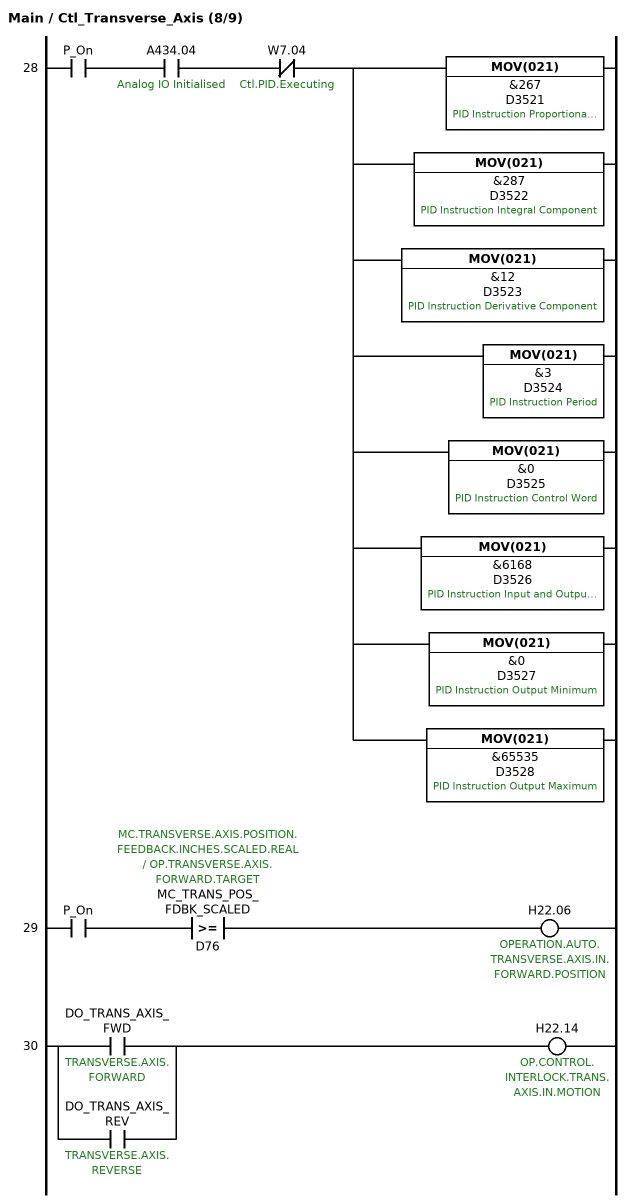
; rung 28
LD P_On
AND A434.04  ; Analog IO Initialised
ANDNOT W7.04  ; Ctl.PID.Executing
MOV(021) &267 D3521  ; PID Instruction Proportional Component
MOV(021) &287 D3522  ; PID Instruction Integral Component
MOV(021) &12 D3523  ; PID Instruction Derivative Component
MOV(021) &3 D3524  ; PID Instruction Period
MOV(021) &0 D3525  ; PID Instruction Control Word
MOV(021) &6168 D3526  ; PID Instruction Input and Output Range Setting
MOV(021) &0 D3527  ; PID Instruction Output Minimum
MOV(021) &65535 D3528  ; PID Instruction Output Maximum
; rung 29
LD P_On
AND>=F(334) MC_TRANS_POS_FDBK_SCALED D76  ; MC.TRANSVERSE.AXIS.POSITION.FEEDBACK.INCHES.SCALED.REAL, OP.TRANSVERSE.AXIS.FORWARD.TARGET
OUT H22.06  ; OPERATION.AUTO.TRANSVERSE.AXIS.IN.FORWARD.POSITION
; rung 30
LD DO_TRANS_AXIS_FWD  ; TRANSVERSE.AXIS.FORWARD
OR DO_TRANS_AXIS_REV  ; TRANSVERSE.AXIS.REVERSE
OUT H22.14  ; OP.CONTROL.INTERLOCK.TRANS.AXIS.IN.MOTION

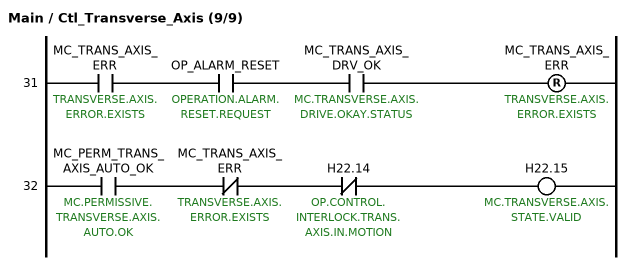
; rung 31
LD MC_TRANS_AXIS_ERR  ; TRANSVERSE.AXIS.ERROR.EXISTS
AND OP_ALARM_RESET  ; OPERATION.ALARM.RESET.REQUEST
AND MC_TRANS_AXIS_DRV_OK  ; MC.TRANSVERSE.AXIS.DRIVE.OKAY.STATUS
RSET MC_TRANS_AXIS_ERR  ; TRANSVERSE.AXIS.ERROR.EXISTS
; rung 32
LD MC_PERM_TRANS_AXIS_AUTO_OK  ; MC.PERMISSIVE.TRANSVERSE.AXIS.AUTO.OK
ANDNOT MC_TRANS_AXIS_ERR  ; TRANSVERSE.AXIS.ERROR.EXISTS
ANDNOT H22.14  ; OP.CONTROL.INTERLOCK.TRANS.AXIS.IN.MOTION
OUT H22.15  ; MC.TRANSVERSE.AXIS.STATE.VALID

### Section Ctl_Saw

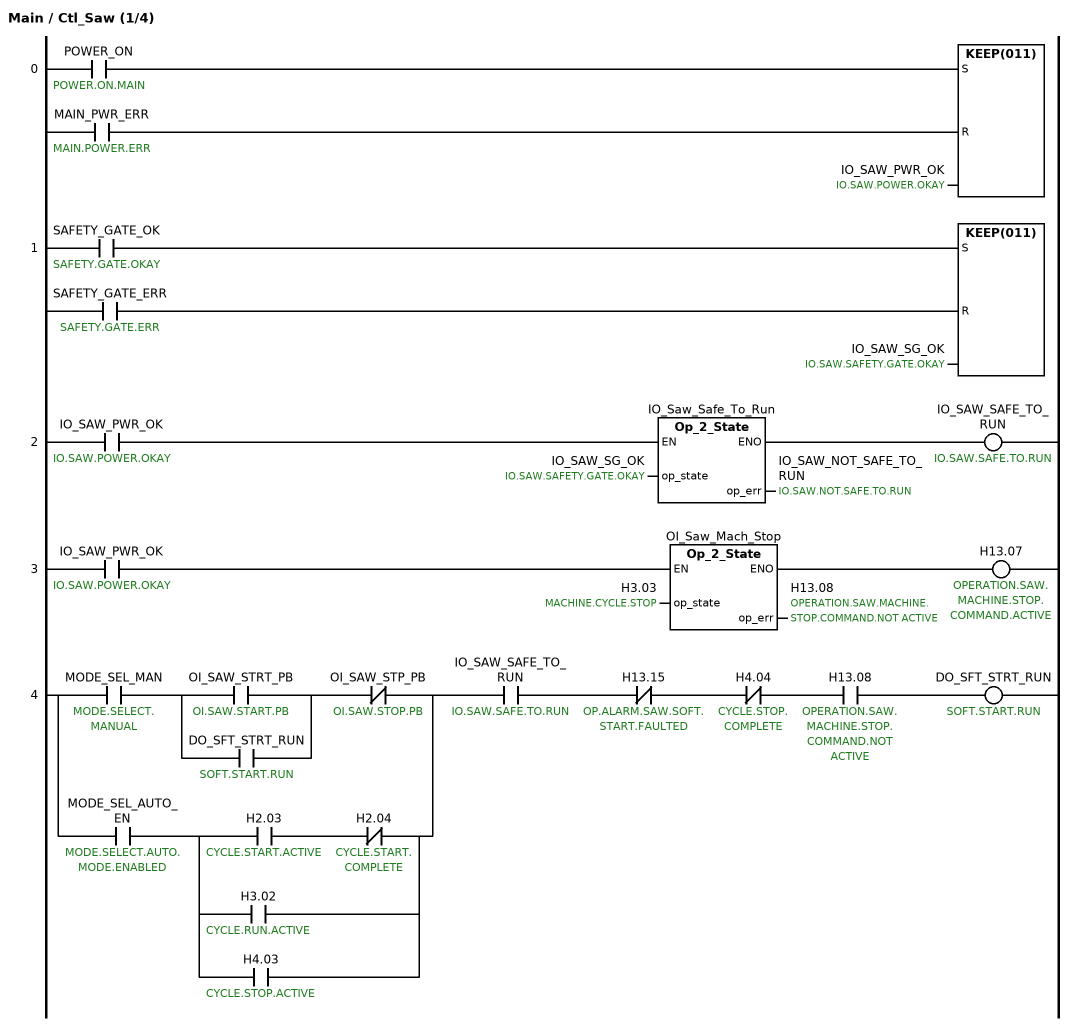
; rung 0
LD POWER_ON  ; POWER.ON.MAIN
LD MAIN_PWR_ERR  ; MAIN.POWER.ERR
KEEP(011) IO_SAW_PWR_OK  ; IO.SAW.POWER.OKAY
; rung 1
LD SAFETY_GATE_OK  ; SAFETY.GATE.OKAY
LD SAFETY_GATE_ERR  ; SAFETY.GATE.ERR
KEEP(011) IO_SAW_SG_OK  ; IO.SAW.SAFETY.GATE.OKAY
; rung 2
LD IO_SAW_PWR_OK  ; IO.SAW.POWER.OKAY
CALL IO_Saw_Safe_To_Run : Op_2_State (op_state := IO_SAW_SG_OK, op_err => IO_SAW_NOT_SAFE_TO_RUN)  ; IO.SAW.SAFETY.GATE.OKAY, IO.SAW.NOT.SAFE.TO.RUN
OUT IO_SAW_SAFE_TO_RUN  ; IO.SAW.SAFE.TO.RUN
; rung 3
LD IO_SAW_PWR_OK  ; IO.SAW.POWER.OKAY
CALL OI_Saw_Mach_Stop : Op_2_State (op_state := H3.03, op_err => H13.08)  ; MACHINE.CYCLE.STOP, OPERATION.SAW.MACHINE.STOP.COMMAND.NOT ACTIVE
OUT H13.07  ; OPERATION.SAW.MACHINE.STOP.COMMAND.ACTIVE
; rung 4
LD MODE_SEL_MAN  ; MODE.SELECT.MANUAL
LD OI_SAW_STRT_PB  ; OI.SAW.START.PB
OR DO_SFT_STRT_RUN  ; SOFT.START.RUN
ANDLD
ANDNOT OI_SAW_STP_PB  ; OI.SAW.STOP.PB
LD MODE_SEL_AUTO_EN  ; MODE.SELECT.AUTO.MODE.ENABLED
LD H2.03  ; CYCLE.START.ACTIVE
ANDNOT H2.04  ; CYCLE.START.COMPLETE
OR H3.02  ; CYCLE.RUN.ACTIVE
OR H4.03  ; CYCLE.STOP.ACTIVE
ANDLD
ORLD
AND IO_SAW_SAFE_TO_RUN  ; IO.SAW.SAFE.TO.RUN
ANDNOT H13.15  ; OP.ALARM.SAW.SOFT.START.FAULTED
ANDNOT H4.04  ; CYCLE.STOP.COMPLETE
AND H13.08  ; OPERATION.SAW.MACHINE.STOP.COMMAND.NOT ACTIVE
OUT DO_SFT_STRT_RUN  ; SOFT.START.RUN

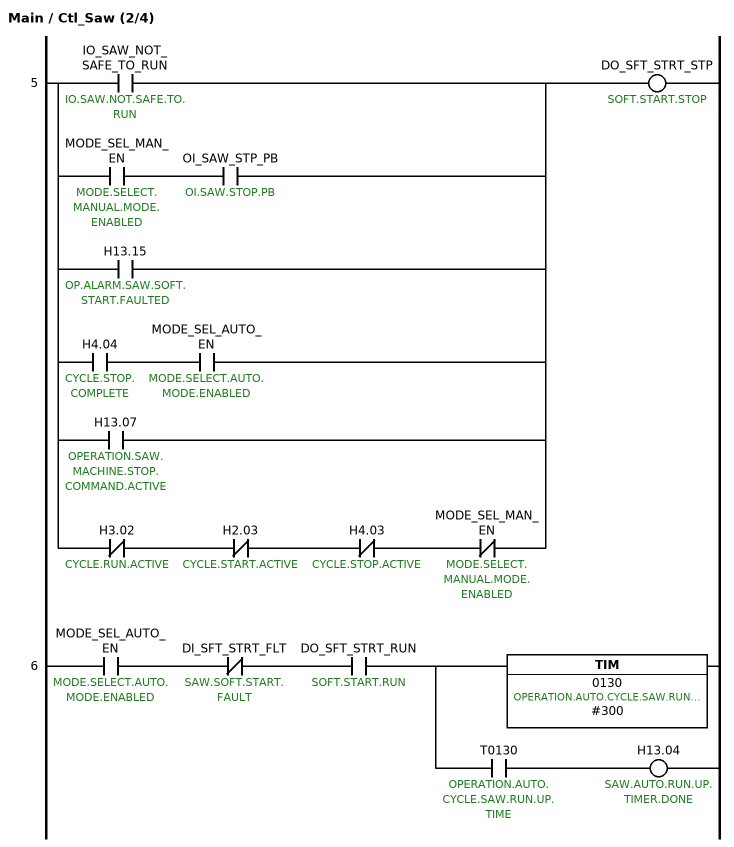
; rung 5
LD IO_SAW_NOT_SAFE_TO_RUN  ; IO.SAW.NOT.SAFE.TO.RUN
LD MODE_SEL_MAN_EN  ; MODE.SELECT.MANUAL.MODE.ENABLED
AND OI_SAW_STP_PB  ; OI.SAW.STOP.PB
ORLD
OR H13.15  ; OP.ALARM.SAW.SOFT.START.FAULTED
LD H4.04  ; CYCLE.STOP.COMPLETE
AND MODE_SEL_AUTO_EN  ; MODE.SELECT.AUTO.MODE.ENABLED
ORLD
OR H13.07  ; OPERATION.SAW.MACHINE.STOP.COMMAND.ACTIVE
LDNOT H3.02  ; CYCLE.RUN.ACTIVE
ANDNOT H2.03  ; CYCLE.START.ACTIVE
ANDNOT H4.03  ; CYCLE.STOP.ACTIVE
ANDNOT MODE_SEL_MAN_EN  ; MODE.SELECT.MANUAL.MODE.ENABLED
ORLD
OUT DO_SFT_STRT_STP  ; SOFT.START.STOP
; rung 6
LD MODE_SEL_AUTO_EN  ; MODE.SELECT.AUTO.MODE.ENABLED
ANDNOT DI_SFT_STRT_FLT  ; SAW.SOFT.START.FAULT
AND DO_SFT_STRT_RUN  ; SOFT.START.RUN
TIM 0130 #300  ; OPERATION.AUTO.CYCLE.SAW.RUN.UP.TIME
AND T0130  ; OPERATION.AUTO.CYCLE.SAW.RUN.UP.TIME
OUT H13.04  ; SAW.AUTO.RUN.UP.TIMER.DONE

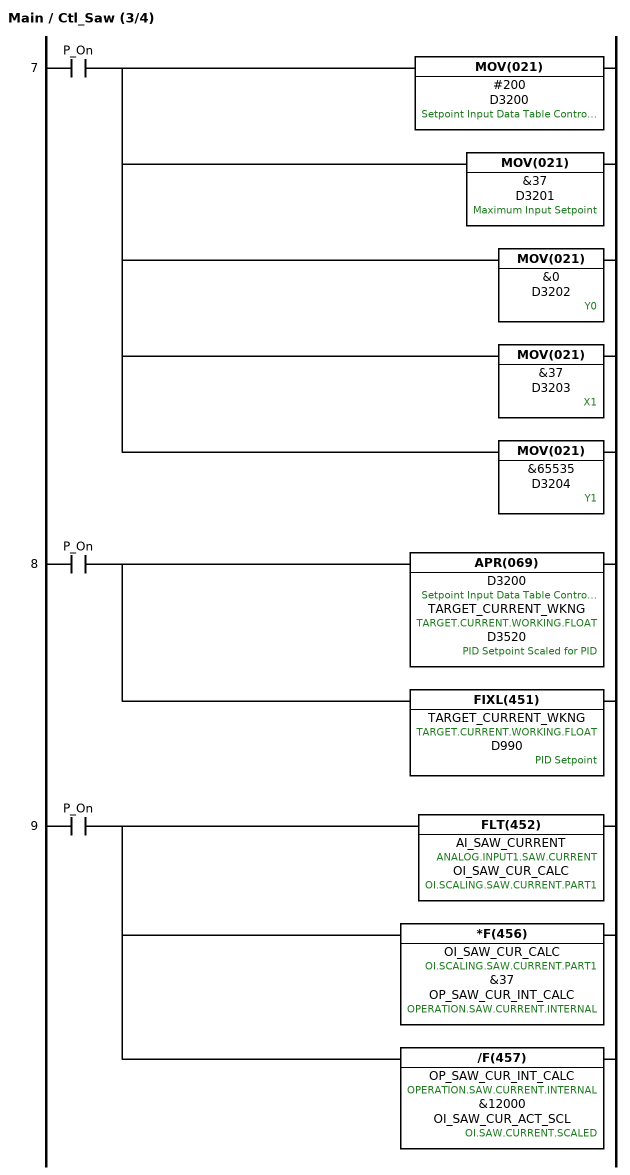
; rung 7
LD P_On
MOV(021) #200 D3200  ; Setpoint Input Data Table Control Word
MOV(021) &37 D3201  ; Maximum Input Setpoint
MOV(021) &0 D3202  ; Y0
MOV(021) &37 D3203  ; X1
MOV(021) &65535 D3204  ; Y1
; rung 8
LD P_On
APR(069) D3200 TARGET_CURRENT_WKNG D3520  ; Setpoint Input Data Table Control Word, TARGET.CURRENT.WORKING.FLOAT, PID Setpoint Scaled for PID
FIXL(451) TARGET_CURRENT_WKNG D990  ; TARGET.CURRENT.WORKING.FLOAT, PID Setpoint
; rung 9
LD P_On
FLT(452) AI_SAW_CURRENT OI_SAW_CUR_CALC  ; ANALOG.INPUT1.SAW.CURRENT, OI.SCALING.SAW.CURRENT.PART1
*F(456) OI_SAW_CUR_CALC &37 OP_SAW_CUR_INT_CALC  ; OI.SCALING.SAW.CURRENT.PART1, OPERATION.SAW.CURRENT.INTERNAL
/F(457) OP_SAW_CUR_INT_CALC &12000 OI_SAW_CUR_ACT_SCL  ; OPERATION.SAW.CURRENT.INTERNAL, OI.SAW.CURRENT.SCALED

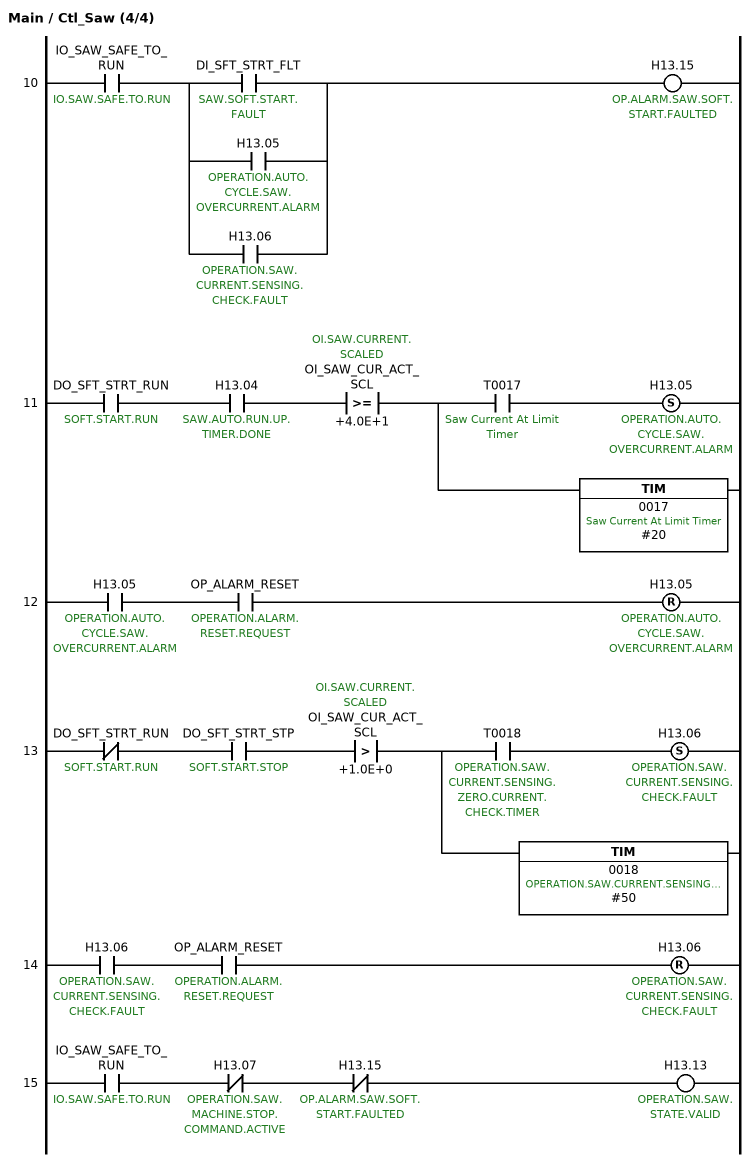
; rung 10
LD IO_SAW_SAFE_TO_RUN  ; IO.SAW.SAFE.TO.RUN
LD DI_SFT_STRT_FLT  ; SAW.SOFT.START.FAULT
OR H13.05  ; OPERATION.AUTO.CYCLE.SAW.OVERCURRENT.ALARM
OR H13.06  ; OPERATION.SAW.CURRENT.SENSING.CHECK.FAULT
ANDLD
OUT H13.15  ; OP.ALARM.SAW.SOFT.START.FAULTED
; rung 11
LD DO_SFT_STRT_RUN  ; SOFT.START.RUN
AND H13.04  ; SAW.AUTO.RUN.UP.TIMER.DONE
AND>=F(334) OI_SAW_CUR_ACT_SCL +4.0E+1  ; OI.SAW.CURRENT.SCALED
OUT TR0
AND T0017  ; Saw Current At Limit Timer
SET H13.05  ; OPERATION.AUTO.CYCLE.SAW.OVERCURRENT.ALARM
LD TR0
TIM 0017 #20  ; Saw Current At Limit Timer
; rung 12
LD H13.05  ; OPERATION.AUTO.CYCLE.SAW.OVERCURRENT.ALARM
AND OP_ALARM_RESET  ; OPERATION.ALARM.RESET.REQUEST
RSET H13.05  ; OPERATION.AUTO.CYCLE.SAW.OVERCURRENT.ALARM
; rung 13
LDNOT DO_SFT_STRT_RUN  ; SOFT.START.RUN
AND DO_SFT_STRT_STP  ; SOFT.START.STOP
AND>F(333) OI_SAW_CUR_ACT_SCL +1.0E+0  ; OI.SAW.CURRENT.SCALED
OUT TR0
AND T0018  ; OPERATION.SAW.CURRENT.SENSING.ZERO.CURRENT.CHECK.TIMER
SET H13.06  ; OPERATION.SAW.CURRENT.SENSING.CHECK.FAULT
LD TR0
TIM 0018 #50  ; OPERATION.SAW.CURRENT.SENSING.ZERO.CURRENT.CHECK.TIMER
; rung 14
LD H13.06  ; OPERATION.SAW.CURRENT.SENSING.CHECK.FAULT
AND OP_ALARM_RESET  ; OPERATION.ALARM.RESET.REQUEST
RSET H13.06  ; OPERATION.SAW.CURRENT.SENSING.CHECK.FAULT
; rung 15
LD IO_SAW_SAFE_TO_RUN  ; IO.SAW.SAFE.TO.RUN
ANDNOT H13.07  ; OPERATION.SAW.MACHINE.STOP.COMMAND.ACTIVE
ANDNOT H13.15  ; OP.ALARM.SAW.SOFT.START.FAULTED
OUT H13.13  ; OPERATION.SAW.STATE.VALID

### Section Ctl_Water

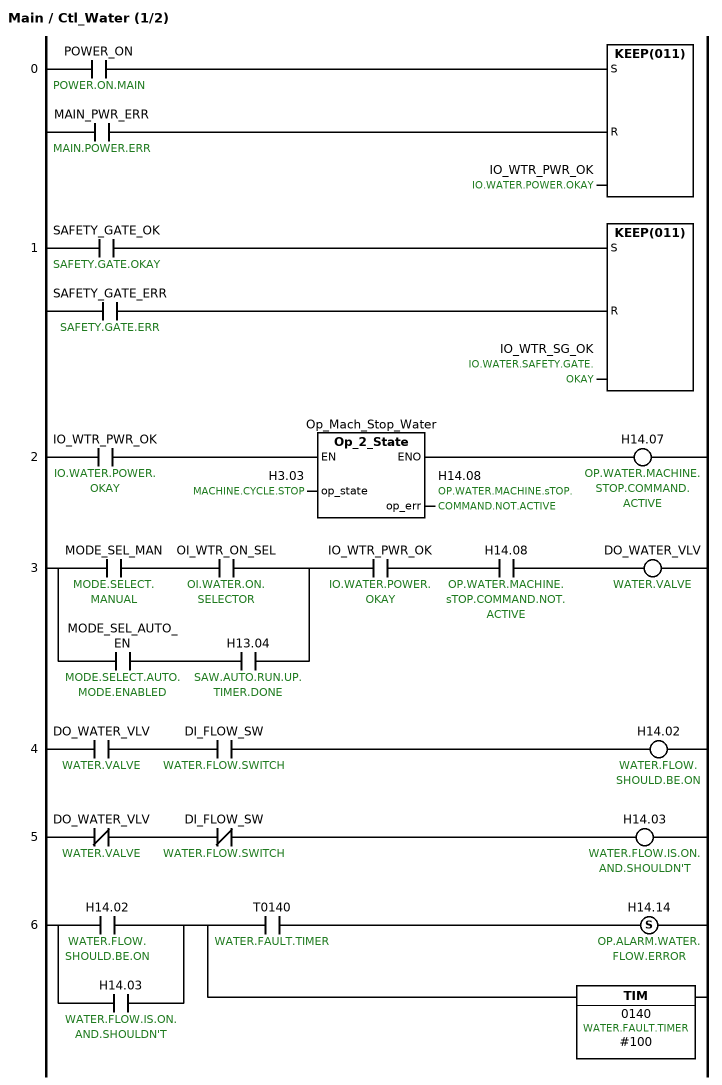
; rung 0
LD POWER_ON  ; POWER.ON.MAIN
LD MAIN_PWR_ERR  ; MAIN.POWER.ERR
KEEP(011) IO_WTR_PWR_OK  ; IO.WATER.POWER.OKAY
; rung 1
LD SAFETY_GATE_OK  ; SAFETY.GATE.OKAY
LD SAFETY_GATE_ERR  ; SAFETY.GATE.ERR
KEEP(011) IO_WTR_SG_OK  ; IO.WATER.SAFETY.GATE.OKAY
; rung 2
LD IO_WTR_PWR_OK  ; IO.WATER.POWER.OKAY
CALL Op_Mach_Stop_Water : Op_2_State (op_state := H3.03, op_err => H14.08)  ; MACHINE.CYCLE.STOP, OP.WATER.MACHINE.sTOP.COMMAND.NOT.ACTIVE
OUT H14.07  ; OP.WATER.MACHINE.STOP.COMMAND.ACTIVE
; rung 3
LD MODE_SEL_MAN  ; MODE.SELECT.MANUAL
AND OI_WTR_ON_SEL  ; OI.WATER.ON.SELECTOR
LD MODE_SEL_AUTO_EN  ; MODE.SELECT.AUTO.MODE.ENABLED
AND H13.04  ; SAW.AUTO.RUN.UP.TIMER.DONE
ORLD
AND IO_WTR_PWR_OK  ; IO.WATER.POWER.OKAY
AND H14.08  ; OP.WATER.MACHINE.sTOP.COMMAND.NOT.ACTIVE
OUT DO_WATER_VLV  ; WATER.VALVE
; rung 4
LD DO_WATER_VLV  ; WATER.VALVE
AND DI_FLOW_SW  ; WATER.FLOW.SWITCH
OUT H14.02  ; WATER.FLOW.SHOULD.BE.ON
; rung 5
LDNOT DO_WATER_VLV  ; WATER.VALVE
ANDNOT DI_FLOW_SW  ; WATER.FLOW.SWITCH
OUT H14.03  ; WATER.FLOW.IS.ON.AND.SHOULDN'T
; rung 6
LD H14.02  ; WATER.FLOW.SHOULD.BE.ON
OR H14.03  ; WATER.FLOW.IS.ON.AND.SHOULDN'T
OUT TR0
AND T0140  ; WATER.FAULT.TIMER
SET H14.14  ; OP.ALARM.WATER.FLOW.ERROR
LD TR0
TIM 0140 #100  ; WATER.FAULT.TIMER

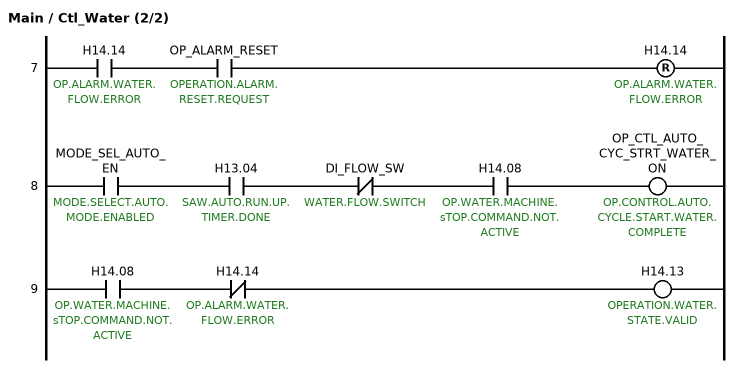
; rung 7
LD H14.14  ; OP.ALARM.WATER.FLOW.ERROR
AND OP_ALARM_RESET  ; OPERATION.ALARM.RESET.REQUEST
RSET H14.14  ; OP.ALARM.WATER.FLOW.ERROR
; rung 8
LD MODE_SEL_AUTO_EN  ; MODE.SELECT.AUTO.MODE.ENABLED
AND H13.04  ; SAW.AUTO.RUN.UP.TIMER.DONE
ANDNOT DI_FLOW_SW  ; WATER.FLOW.SWITCH
AND H14.08  ; OP.WATER.MACHINE.sTOP.COMMAND.NOT.ACTIVE
OUT OP_CTL_AUTO_CYC_STRT_WATER_ON  ; OP.CONTROL.AUTO.CYCLE.START.WATER.COMPLETE
; rung 9
LD H14.08  ; OP.WATER.MACHINE.sTOP.COMMAND.NOT.ACTIVE
ANDNOT H14.14  ; OP.ALARM.WATER.FLOW.ERROR
OUT H14.13  ; OPERATION.WATER.STATE.VALID

### Section Ctl_Lazer

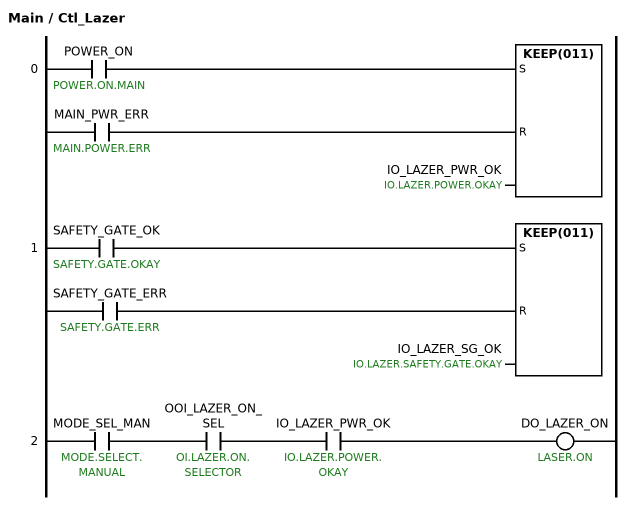
; rung 0
LD POWER_ON  ; POWER.ON.MAIN
LD MAIN_PWR_ERR  ; MAIN.POWER.ERR
KEEP(011) IO_LAZER_PWR_OK  ; IO.LAZER.POWER.OKAY
; rung 1
LD SAFETY_GATE_OK  ; SAFETY.GATE.OKAY
LD SAFETY_GATE_ERR  ; SAFETY.GATE.ERR
KEEP(011) IO_LAZER_SG_OK  ; IO.LAZER.SAFETY.GATE.OKAY
; rung 2
LD MODE_SEL_MAN  ; MODE.SELECT.MANUAL
AND OOI_LAZER_ON_SEL  ; OI.LAZER.ON.SELECTOR
AND IO_LAZER_PWR_OK  ; IO.LAZER.POWER.OKAY
OUT DO_LAZER_ON  ; LASER.ON

### Section Init_Recipe

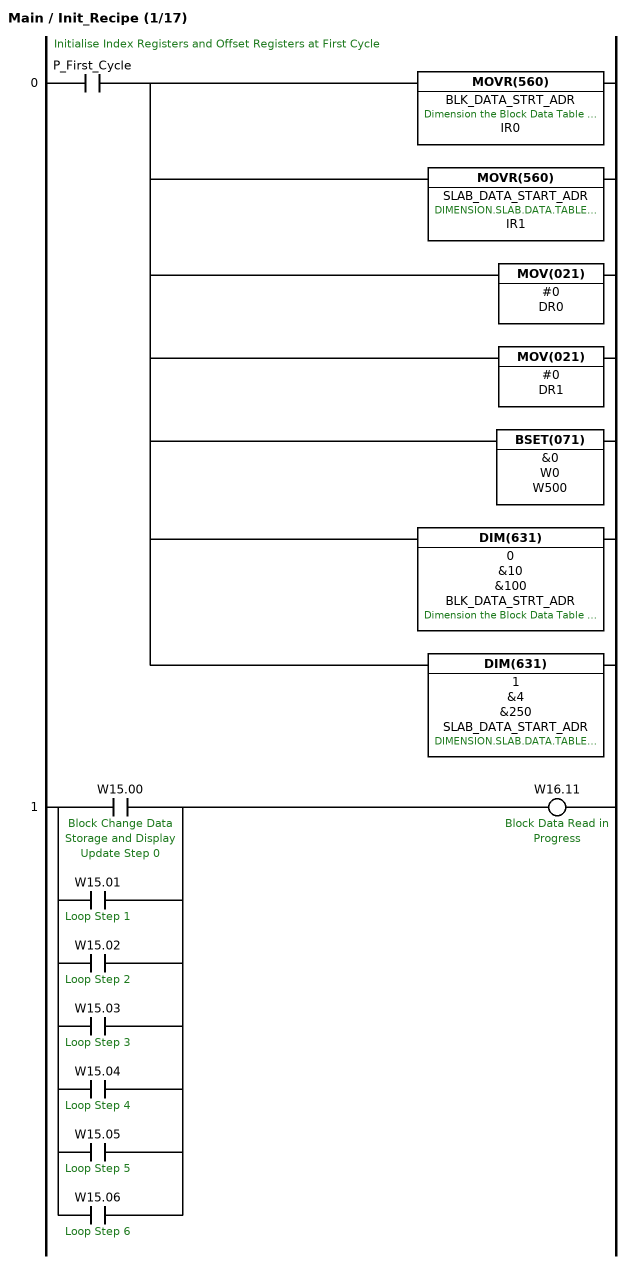
; rung 0: Initialise Index Registers and Offset Registers at First Cycle
LD P_First_Cycle
MOVR(560) BLK_DATA_STRT_ADR IR0  ; Dimension the Block Data Table - Start Address
MOVR(560) SLAB_DATA_START_ADR IR1  ; DIMENSION.SLAB.DATA.TABLE.START.ADDRESS
MOV(021) #0 DR0
MOV(021) #0 DR1
BSET(071) &0 W0 W500
DIM(631) 0 &10 &100 BLK_DATA_STRT_ADR  ; Dimension the Block Data Table - Start Address
DIM(631) 1 &4 &250 SLAB_DATA_START_ADR  ; DIMENSION.SLAB.DATA.TABLE.START.ADDRESS
; rung 1
LD W15.00  ; Block Change Data Storage and Display Update Step 0
OR W15.01  ; Loop Step 1
OR W15.02  ; Loop Step 2
OR W15.03  ; Loop Step 3
OR W15.04  ; Loop Step 4
OR W15.05  ; Loop Step 5
OR W15.06  ; Loop Step 6
OUT W16.11  ; Block Data Read in Progress

